LIN {X 0.136,Y -541.302,Z 1152.951,A 0.000,B 0.000,C 90.000,E1 27.078} C_DIS
LIN {X 0.205,Y -536.132,Z 1152.947,A 0.000,B 0.000,C 90.000,E1 26.360} C_DIS
LIN {X 0.131,Y -531.673,Z 1152.943,A 0.000,B 0.000,C 90.000,E1 25.796} C_DIS
LIN {X 0.041,Y -524.620,Z 1152.939,A 0.000,B 0.000,C 90.000,E1 24.951} C_DIS
LIN {X -0.042,Y -515.804,Z 1152.933,A 0.000,B 0.000,C 90.000,E1 23.951} C_DIS
LIN {X -0.075,Y -509.279,Z 1152.929,A 0.000,B 0.000,C 90.000,E1 23.259} C_DIS
LIN {X -0.034,Y -503.804,Z 1152.926,A 0.000,B 0.000,C 90.000,E1 22.695} C_DIS
LIN {X -0.151,Y -492.766,Z 1152.920,A 0.000,B 0.000,C 90.000,E1 21.642} C_DIS
LIN {X -0.103,Y -481.579,Z 1152.914,A 0.000,B 0.000,C 90.000,E1 20.610} C_DIS
LIN {X -0.257,Y -469.838,Z 1152.909,A 0.000,B 0.000,C 90.000,E1 19.577} C_DIS
LIN {X -0.031,Y -457.925,Z 1152.903,A 0.000,B 0.000,C 90.000,E1 18.489} C_DIS
LIN {X -0.234,Y -435.893,Z 1152.891,A 0.000,B 0.000,C 90.000,E1 16.441} C_DIS
LIN {X 0.046,Y -423.104,Z 1152.884,A 0.000,B 0.000,C 90.000,E1 15.064} C_DIS
LIN {X 0.162,Y -412.046,Z 1152.877,A 0.000,B 0.000,C 90.000,E1 13.772} C_DIS
LIN {X 0.036,Y -404.119,Z 1152.871,A 0.000,B 0.000,C 90.000,E1 12.771} C_DIS
LIN {X 0.073,Y -398.095,Z 1152.866,A 0.000,B 0.000,C 90.000,E1 11.895} C_DIS
LIN {X 0.107,Y -396.971,Z 1152.865,A 0.000,B 0.000,C 90.000,E1 11.715} C_DIS
LIN {X -0.009,Y -393.901,Z 1152.862,A 0.000,B 0.000,C 90.000,E1 11.130} C_DIS
LIN {X -0.016,Y -392.561,Z 1152.860,A 0.000,B 0.000,C 90.000,E1 10.715} C_DIS
LIN {X -0.198,Y -392.478,Z 1152.857,A 0.000,B 0.000,C 90.000,E1 10.254} C_DIS
LIN {X 0.110,Y -393.719,Z 1152.853,A 0.000,B 0.000,C 90.000,E1 9.500} C_DIS
LIN {X 0.046,Y -396.236,Z 1152.848,A 0.000,B 0.000,C 90.000,E1 8.624} C_DIS
LIN {X -0.148,Y -401.677,Z 1152.839,A 0.000,B 0.000,C 90.000,E1 7.068} C_DIS
LIN {X -0.013,Y -405.388,Z 1152.835,A 0.000,B 0.000,C 90.000,E1 6.258} C_DIS
LIN {X -0.013,Y -407.563,Z 1152.833,A 0.000,B 0.000,C 90.000,E1 5.910} C_DIS
LIN {X -0.080,Y -410.731,Z 1152.831,A 0.000,B 0.000,C 90.000,E1 5.568} C_DIS
LIN {X 0.043,Y -412.332,Z 1152.830,A 0.000,B 0.000,C 90.000,E1 5.391} C_DIS
LIN {X -0.036,Y -437.093,Z 1152.820,A 0.000,B 0.000,C 90.000,E1 3.555} C_DIS
LIN {X 0.076,Y -456.596,Z 1152.812,A 0.000,B 0.000,C 90.000,E1 2.178} C_DIS
LIN {X -0.104,Y -467.873,Z 1152.808,A 0.000,B 0.000,C 90.000,E1 1.432} C_DIS
LIN {X -0.166,Y -477.392,Z 1152.804,A 0.000,B 0.000,C 90.000,E1 0.802} C_DIS
LIN {X 0.000,Y -488.031,Z 1152.800,A 0.000,B 0.000,C 90.000,E1 360.000} C_DIS
LIN {X 0.105,Y -495.261,Z 1152.797,A 0.000,B 0.000,C 90.000,E1 359.427} C_DIS
LIN {X -0.233,Y -502.565,Z 1152.794,A 0.000,B 0.000,C 90.000,E1 358.854} C_DIS
LIN {X 0.184,Y -509.593,Z 1152.790,A 0.000,B 0.000,C 90.000,E1 358.165} C_DIS
LIN {X 0.238,Y -516.287,Z 1152.786,A 0.000,B 0.000,C 90.000,E1 357.478} C_DIS
LIN {X 0.222,Y -522.608,Z 1152.782,A 0.000,B 0.000,C 90.000,E1 356.788} C_DIS
LIN {X 0.006,Y -528.517,Z 1152.778,A 0.000,B 0.000,C 90.000,E1 356.102} C_DIS
LIN {X -0.016,Y -532.952,Z 1152.775,A 0.000,B 0.000,C 90.000,E1 355.527} C_DIS
LIN {X -0.273,Y -537.881,Z 1152.771,A 0.000,B 0.000,C 90.000,E1 354.837} C_DIS
LIN {X 0.047,Y -542.345,Z 1152.767,A 0.000,B 0.000,C 90.000,E1 354.090} C_DIS
LIN {X 0.129,Y -545.610,Z 1152.764,A 0.000,B 0.000,C 90.000,E1 353.514} C_DIS
LIN {X -0.217,Y -549.964,Z 1152.759,A 0.000,B 0.000,C 90.000,E1 352.704} C_DIS
LIN {X 0.176,Y -552.026,Z 1152.757,A 0.000,B 0.000,C 90.000,E1 352.243} C_DIS
LIN {X 0.150,Y -555.072,Z 1152.753,A 0.000,B 0.000,C 90.000,E1 351.546} C_DIS
LIN {X -0.102,Y -558.385,Z 1152.749,A 0.000,B 0.000,C 90.000,E1 350.735} C_DIS
LIN {X -0.228,Y -561.402,Z 1152.744,A 0.000,B 0.000,C 90.000,E1 349.916} C_DIS
LIN {X -0.261,Y -564.948,Z 1152.738,A 0.000,B 0.000,C 90.000,E1 348.814} C_DIS
LIN {X 0.241,Y -567.386,Z 1152.733,A 0.000,B 0.000,C 90.000,E1 347.937} C_DIS
LIN {X -0.158,Y -570.402,Z 1152.727,A 0.000,B 0.000,C 90.000,E1 346.881} C_DIS
LIN {X -0.189,Y -573.924,Z 1152.719,A 0.000,B 0.000,C 90.000,E1 345.519} C_DIS
LIN {X 0.197,Y -576.570,Z 1152.714,A 0.000,B 0.000,C 90.000,E1 344.393} C_DIS
LIN {X 0.061,Y -579.116,Z 1152.707,A 0.000,B 0.000,C 90.000,E1 343.323} C_DIS
LIN {X 0.129,Y -581.561,Z 1152.701,A 0.000,B 0.000,C 90.000,E1 342.236} C_DIS
LIN {X 0.236,Y -583.874,Z 1152.695,A 0.000,B 0.000,C 90.000,E1 341.148} C_DIS
LIN {X -0.178,Y -585.938,Z 1152.689,A 0.000,B 0.000,C 90.000,E1 340.115} C_DIS
LIN {X 0.319,Y -587.363,Z 1152.685,A 0.000,B 0.000,C 90.000,E1 339.263} C_DIS
LIN {X -0.179,Y -589.454,Z 1152.678,A 0.000,B 0.000,C 90.000,E1 337.975} C_DIS
LIN {X -0.202,Y -590.421,Z 1152.673,A 0.000,B 0.000,C 90.000,E1 337.177} C_DIS
LIN {X 0.343,Y -591.464,Z 1152.666,A 0.000,B 0.000,C 90.000,E1 335.793} C_DIS
LIN {X -0.210,Y -591.834,Z 1152.661,A 0.000,B 0.000,C 90.000,E1 335.049} C_DIS
LIN {X 0.020,Y -591.879,Z 1152.657,A 0.000,B 0.000,C 90.000,E1 334.229} C_DIS
LIN {X 0.081,Y -591.762,Z 1152.654,A 0.000,B 0.000,C 90.000,E1 333.691} C_DIS
LIN {X 0.312,Y -591.168,Z 1152.650,A 0.000,B 0.000,C 90.000,E1 332.871} C_DIS
LIN {X 0.108,Y -590.627,Z 1152.647,A 0.000,B 0.000,C 90.000,E1 332.359} C_DIS
LIN {X 0.073,Y -589.543,Z 1152.642,A 0.000,B 0.000,C 90.000,E1 331.563} C_DIS
LIN {X -0.252,Y -588.050,Z 1152.638,A 0.000,B 0.000,C 90.000,E1 330.795} C_DIS
LIN {X -0.190,Y -586.837,Z 1152.635,A 0.000,B 0.000,C 90.000,E1 330.255} C_DIS
LIN {X 0.248,Y -584.613,Z 1152.630,A 0.000,B 0.000,C 90.000,E1 329.410} C_DIS
LIN {X 0.153,Y -581.952,Z 1152.626,A 0.000,B 0.000,C 90.000,E1 328.614} C_DIS
LIN {X 0.101,Y -579.167,Z 1152.622,A 0.000,B 0.000,C 90.000,E1 327.946} C_DIS
LIN {X 0.330,Y -575.786,Z 1152.618,A 0.000,B 0.000,C 90.000,E1 327.248} C_DIS
LIN {X -0.262,Y -571.745,Z 1152.615,A 0.000,B 0.000,C 90.000,E1 326.628} C_DIS
LIN {X -0.089,Y -567.295,Z 1152.611,A 0.000,B 0.000,C 90.000,E1 325.928} C_DIS
LIN {X -0.172,Y -563.456,Z 1152.608,A 0.000,B 0.000,C 90.000,E1 325.388} C_DIS
LIN {X 0.037,Y -559.163,Z 1152.605,A 0.000,B 0.000,C 90.000,E1 324.815} C_DIS
LIN {X -0.074,Y -551.011,Z 1152.599,A 0.000,B 0.000,C 90.000,E1 323.863} C_DIS
LIN {X 0.078,Y -546.038,Z 1152.596,A 0.000,B 0.000,C 90.000,E1 323.290} C_DIS
LIN {X 0.151,Y -530.643,Z 1152.587,A 0.000,B 0.000,C 90.000,E1 321.618} C_DIS
LIN {X 0.220,Y -526.479,Z 1152.584,A 0.000,B 0.000,C 90.000,E1 321.090} C_DIS
LIN {X 0.001,Y -523.789,Z 1152.581,A 0.000,B 0.000,C 90.000,E1 320.642} C_DIS
LIN {X -0.080,Y -521.477,Z 1152.578,A 0.000,B 0.000,C 90.000,E1 320.070} C_DIS
LIN {X 0.155,Y -520.483,Z 1152.575,A 0.000,B 0.000,C 90.000,E1 319.461} C_DIS
LIN {X -0.167,Y -520.045,Z 1152.570,A 0.000,B 0.000,C 90.000,E1 318.566} C_DIS
LIN {X 0.178,Y -520.307,Z 1152.562,A 0.000,B 0.000,C 90.000,E1 317.067} C_DIS
LIN {X 0.017,Y -521.216,Z 1152.550,A 0.000,B 0.000,C 90.000,E1 315.040} C_DIS
LIN {X 0.024,Y -521.900,Z 1152.542,A 0.000,B 0.000,C 90.000,E1 313.581} C_DIS
LIN {X -0.080,Y -522.795,Z 1152.531,A 0.000,B 0.000,C 90.000,E1 311.553} C_DIS
LIN {X -0.074,Y -523.671,Z 1152.521,A 0.000,B 0.000,C 90.000,E1 309.806} C_DIS
LIN {X 0.307,Y -524.813,Z 1152.510,A 0.000,B 0.000,C 90.000,E1 307.729} C_DIS
LIN {X 0.133,Y -525.768,Z 1152.502,A 0.000,B 0.000,C 90.000,E1 306.297} C_DIS
LIN {X 0.070,Y -526.827,Z 1152.492,A 0.000,B 0.000,C 90.000,E1 304.565} C_DIS
LIN {X 0.067,Y -527.667,Z 1152.484,A 0.000,B 0.000,C 90.000,E1 303.118} C_DIS
LIN {X 0.039,Y -528.892,Z 1152.474,A 0.000,B 0.000,C 90.000,E1 301.386} C_DIS
LIN {X -0.075,Y -530.043,Z 1152.465,A 0.000,B 0.000,C 90.000,E1 299.667} C_DIS
LIN {X -0.250,Y -530.572,Z 1152.460,A 0.000,B 0.000,C 90.000,E1 298.821} C_DIS
LIN {X 0.182,Y -531.222,Z 1152.452,A 0.000,B 0.000,C 90.000,E1 297.334} C_DIS
LIN {X -0.087,Y -531.533,Z 1152.444,A 0.000,B 0.000,C 90.000,E1 295.924} C_DIS
LIN {X 0.126,Y -531.679,Z 1152.436,A 0.000,B 0.000,C 90.000,E1 294.463} C_DIS
LIN {X -0.178,Y -531.663,Z 1152.426,A 0.000,B 0.000,C 90.000,E1 292.770} C_DIS
LIN {X -0.195,Y -531.621,Z 1152.417,A 0.000,B 0.000,C 90.000,E1 291.046} C_DIS
LIN {X 0.089,Y -531.329,Z 1152.409,A 0.000,B 0.000,C 90.000,E1 289.577} C_DIS
LIN {X 0.170,Y -531.006,Z 1152.402,A 0.000,B 0.000,C 90.000,E1 288.417} C_DIS
LIN {X 0.100,Y -530.507,Z 1152.394,A 0.000,B 0.000,C 90.000,E1 286.985} C_DIS
LIN {X 0.198,Y -529.697,Z 1152.385,A 0.000,B 0.000,C 90.000,E1 285.245} C_DIS
LIN {X -0.003,Y -528.817,Z 1152.375,A 0.000,B 0.000,C 90.000,E1 283.536} C_DIS
LIN {X 0.265,Y -527.914,Z 1152.367,A 0.000,B 0.000,C 90.000,E1 282.063} C_DIS
LIN {X -0.094,Y -526.828,Z 1152.358,A 0.000,B 0.000,C 90.000,E1 280.366} C_DIS
LIN {X -0.055,Y -525.829,Z 1152.348,A 0.000,B 0.000,C 90.000,E1 278.624} C_DIS
LIN {X -0.167,Y -524.609,Z 1152.337,A 0.000,B 0.000,C 90.000,E1 276.606} C_DIS
LIN {X -0.255,Y -523.900,Z 1152.329,A 0.000,B 0.000,C 90.000,E1 275.163} C_DIS
LIN {X 0.112,Y -523.232,Z 1152.321,A 0.000,B 0.000,C 90.000,E1 273.669} C_DIS
LIN {X -0.128,Y -522.559,Z 1152.311,A 0.000,B 0.000,C 90.000,E1 271.949} C_DIS
LIN {X 0.187,Y -522.008,Z 1152.303,A 0.000,B 0.000,C 90.000,E1 270.458} C_DIS
LIN {X -0.044,Y -521.317,Z 1152.295,A 0.000,B 0.000,C 90.000,E1 269.026} C_DIS
LIN {X 0.245,Y -520.644,Z 1152.286,A 0.000,B 0.000,C 90.000,E1 267.535} C_DIS
LIN {X 0.056,Y -520.109,Z 1152.280,A 0.000,B 0.000,C 90.000,E1 266.388} C_DIS
LIN {X -0.083,Y -519.632,Z 1152.275,A 0.000,B 0.000,C 90.000,E1 265.527} C_DIS
LIN {X -0.248,Y -518.752,Z 1152.269,A 0.000,B 0.000,C 90.000,E1 264.375} C_DIS
LIN {X 0.089,Y -517.672,Z 1152.262,A 0.000,B 0.000,C 90.000,E1 263.166} C_DIS
LIN {X -0.132,Y -516.199,Z 1152.254,A 0.000,B 0.000,C 90.000,E1 261.724} C_DIS
LIN {X 0.200,Y -514.754,Z 1152.246,A 0.000,B 0.000,C 90.000,E1 260.218} C_DIS
LIN {X 0.008,Y -512.461,Z 1152.233,A 0.000,B 0.000,C 90.000,E1 257.881} C_DIS
LIN {X -0.018,Y -510.366,Z 1152.220,A 0.000,B 0.000,C 90.000,E1 255.519} C_DIS
LIN {X -0.010,Y -508.806,Z 1152.210,A 0.000,B 0.000,C 90.000,E1 253.740} C_DIS
LIN {X 0.189,Y -506.842,Z 1152.198,A 0.000,B 0.000,C 90.000,E1 251.638} C_DIS
LIN {X -0.162,Y -505.371,Z 1152.190,A 0.000,B 0.000,C 90.000,E1 250.188} C_DIS
LIN {X 0.098,Y -503.879,Z 1152.182,A 0.000,B 0.000,C 90.000,E1 248.666} C_DIS
LIN {X 0.120,Y -501.969,Z 1152.172,A 0.000,B 0.000,C 90.000,E1 246.869} C_DIS
LIN {X 0.161,Y -500.575,Z 1152.165,A 0.000,B 0.000,C 90.000,E1 245.665} C_DIS
LIN {X -0.142,Y -498.177,Z 1152.155,A 0.000,B 0.000,C 90.000,E1 243.896} C_DIS
LIN {X 0.114,Y -496.068,Z 1152.147,A 0.000,B 0.000,C 90.000,E1 242.359} C_DIS
LIN {X 0.149,Y -493.416,Z 1152.136,A 0.000,B 0.000,C 90.000,E1 240.539} C_DIS
LIN {X -0.161,Y -492.074,Z 1152.131,A 0.000,B 0.000,C 90.000,E1 239.665} C_DIS
LIN {X 0.276,Y -489.217,Z 1152.121,A 0.000,B 0.000,C 90.000,E1 237.788} C_DIS
LIN {X -0.179,Y -486.354,Z 1152.111,A 0.000,B 0.000,C 90.000,E1 236.008} C_DIS
LIN {X -0.246,Y -483.970,Z 1152.103,A 0.000,B 0.000,C 90.000,E1 234.482} C_DIS
LIN {X 0.101,Y -482.062,Z 1152.096,A 0.000,B 0.000,C 90.000,E1 233.210} C_DIS
LIN {X -0.054,Y -479.043,Z 1152.085,A 0.000,B 0.000,C 90.000,E1 231.376} C_DIS
LIN {X 0.030,Y -477.540,Z 1152.080,A 0.000,B 0.000,C 90.000,E1 230.436} C_DIS
LIN {X 0.287,Y -474.997,Z 1152.072,A 0.000,B 0.000,C 90.000,E1 228.852} C_DIS
LIN {X 0.139,Y -472.390,Z 1152.063,A 0.000,B 0.000,C 90.000,E1 227.310} C_DIS
LIN {X 0.262,Y -469.805,Z 1152.054,A 0.000,B 0.000,C 90.000,E1 225.729} C_DIS
LIN {X -0.095,Y -462.736,Z 1152.023,A 0.000,B 0.000,C 90.000,E1 220.092} C_DIS
LIN {X 0.011,Y -460.932,Z 1152.010,A 0.000,B 0.000,C 90.000,E1 217.855} C_DIS
LIN {X -0.139,Y -459.348,Z 1151.998,A 0.000,B 0.000,C 90.000,E1 215.644} C_DIS
LIN {X -0.208,Y -457.835,Z 1151.970,A 0.000,B 0.000,C 90.000,E1 210.541} C_DIS
LIN {X -0.011,Y -459.088,Z 1151.950,A 0.000,B 0.000,C 90.000,E1 207.001} C_DIS
LIN {X -0.115,Y -461.535,Z 1151.936,A 0.000,B 0.000,C 90.000,E1 204.463} C_DIS
LIN {X -0.027,Y -466.647,Z 1151.918,A 0.000,B 0.000,C 90.000,E1 201.280} C_DIS
LIN {X -0.169,Y -472.328,Z 1151.904,A 0.000,B 0.000,C 90.000,E1 198.779} C_DIS
LIN {X -0.134,Y -480.238,Z 1151.889,A 0.000,B 0.000,C 90.000,E1 195.969} C_DIS
LIN {X 0.189,Y -487.392,Z 1151.877,A 0.000,B 0.000,C 90.000,E1 193.772} C_DIS
LIN {X -0.058,Y -490.516,Z 1151.872,A 0.000,B 0.000,C 90.000,E1 192.883} C_DIS
LIN {X 0.129,Y -499.143,Z 1151.858,A 0.000,B 0.000,C 90.000,E1 190.433} C_DIS
LIN {X 0.196,Y -505.805,Z 1151.848,A 0.000,B 0.000,C 90.000,E1 188.624} C_DIS
LIN {X 0.252,Y -512.574,Z 1151.838,A 0.000,B 0.000,C 90.000,E1 186.834} C_DIS
LIN {X -0.035,Y -518.168,Z 1151.830,A 0.000,B 0.000,C 90.000,E1 185.391} C_DIS
LIN {X 0.246,Y -523.689,Z 1151.822,A 0.000,B 0.000,C 90.000,E1 183.898} C_DIS
LIN {X 0.077,Y -529.165,Z 1151.814,A 0.000,B 0.000,C 90.000,E1 182.465} C_DIS
LIN {X 0.008,Y -534.623,Z 1151.806,A 0.000,B 0.000,C 90.000,E1 181.031} C_DIS
LIN {X 0.027,Y -540.046,Z 1151.798,A 0.000,B 0.000,C 90.000,E1 179.599} C_DIS
LIN {X 0.159,Y -545.569,Z 1151.790,A 0.000,B 0.000,C 90.000,E1 178.165} C_DIS
LIN {X -0.047,Y -553.223,Z 1151.779,A 0.000,B 0.000,C 90.000,E1 176.216} C_DIS
LIN {X -0.199,Y -558.691,Z 1151.771,A 0.000,B 0.000,C 90.000,E1 174.837} C_DIS
LIN {X -0.108,Y -565.163,Z 1151.762,A 0.000,B 0.000,C 90.000,E1 173.166} C_DIS
LIN {X -0.087,Y -569.507,Z 1151.756,A 0.000,B 0.000,C 90.000,E1 172.064} C_DIS
LIN {X 0.108,Y -574.834,Z 1151.748,A 0.000,B 0.000,C 90.000,E1 170.679} C_DIS
LIN {X -0.301,Y -579.038,Z 1151.742,A 0.000,B 0.000,C 90.000,E1 169.634} C_DIS
LIN {X -0.077,Y -585.318,Z 1151.733,A 0.000,B 0.000,C 90.000,E1 167.993} C_DIS
LIN {X -0.232,Y -589.339,Z 1151.727,A 0.000,B 0.000,C 90.000,E1 166.937} C_DIS
LIN {X -0.335,Y -593.227,Z 1151.721,A 0.000,B 0.000,C 90.000,E1 165.880} C_DIS
LIN {X -0.242,Y -596.951,Z 1151.716,A 0.000,B 0.000,C 90.000,E1 164.810} C_DIS
LIN {X -0.094,Y -600.543,Z 1151.710,A 0.000,B 0.000,C 90.000,E1 163.740} C_DIS
LIN {X 0.005,Y -604.837,Z 1151.702,A 0.000,B 0.000,C 90.000,E1 162.417} C_DIS
LIN {X 0.179,Y -608.947,Z 1151.695,A 0.000,B 0.000,C 90.000,E1 161.094} C_DIS
LIN {X -0.214,Y -613.576,Z 1151.686,A 0.000,B 0.000,C 90.000,E1 159.571} C_DIS
LIN {X -0.240,Y -616.490,Z 1151.681,A 0.000,B 0.000,C 90.000,E1 158.539} C_DIS
LIN {X -0.033,Y -620.714,Z 1151.672,A 0.000,B 0.000,C 90.000,E1 156.975} C_DIS
LIN {X 0.268,Y -624.067,Z 1151.665,A 0.000,B 0.000,C 90.000,E1 155.665} C_DIS
LIN {X 0.051,Y -627.391,Z 1151.658,A 0.000,B 0.000,C 90.000,E1 154.409} C_DIS
LIN {X 0.185,Y -631.130,Z 1151.649,A 0.000,B 0.000,C 90.000,E1 152.871} C_DIS
LIN {X -0.209,Y -634.114,Z 1151.642,A 0.000,B 0.000,C 90.000,E1 151.641} C_DIS
LIN {X 0.307,Y -636.973,Z 1151.635,A 0.000,B 0.000,C 90.000,E1 150.333} C_DIS
LIN {X -0.184,Y -640.156,Z 1151.627,A 0.000,B 0.000,C 90.000,E1 148.869} C_DIS
LIN {X 0.211,Y -642.610,Z 1151.620,A 0.000,B 0.000,C 90.000,E1 147.582} C_DIS
LIN {X 0.110,Y -644.885,Z 1151.613,A 0.000,B 0.000,C 90.000,E1 146.342} C_DIS
LIN {X -0.376,Y -646.684,Z 1151.608,A 0.000,B 0.000,C 90.000,E1 145.388} C_DIS
LIN {X 0.007,Y -649.252,Z 1151.599,A 0.000,B 0.000,C 90.000,E1 143.863} C_DIS
LIN {X 0.225,Y -652.104,Z 1151.590,A 0.000,B 0.000,C 90.000,E1 142.110} C_DIS
LIN {X -0.400,Y -655.191,Z 1151.580,A 0.000,B 0.000,C 90.000,E1 140.436} C_DIS
LIN {X -0.084,Y -658.083,Z 1151.572,A 0.000,B 0.000,C 90.000,E1 138.933} C_DIS
LIN {X -0.207,Y -661.090,Z 1151.564,A 0.000,B 0.000,C 90.000,E1 137.472} C_DIS
LIN {X 0.163,Y -664.972,Z 1151.553,A 0.000,B 0.000,C 90.000,E1 135.486} C_DIS
LIN {X 0.168,Y -669.787,Z 1151.541,A 0.000,B 0.000,C 90.000,E1 133.299} C_DIS
LIN {X 0.291,Y -673.754,Z 1151.531,A 0.000,B 0.000,C 90.000,E1 131.595} C_DIS
LIN {X 0.196,Y -678.990,Z 1151.519,A 0.000,B 0.000,C 90.000,E1 129.439} C_DIS
LIN {X 0.012,Y -682.053,Z 1151.513,A 0.000,B 0.000,C 90.000,E1 128.257} C_DIS
LIN {X -0.133,Y -684.994,Z 1151.506,A 0.000,B 0.000,C 90.000,E1 127.076} C_DIS
LIN {X -0.099,Y -688.042,Z 1151.499,A 0.000,B 0.000,C 90.000,E1 125.884} C_DIS
LIN {X 0.022,Y -691.508,Z 1151.491,A 0.000,B 0.000,C 90.000,E1 124.452} C_DIS
LIN {X -0.230,Y -694.370,Z 1151.485,A 0.000,B 0.000,C 90.000,E1 123.293} C_DIS
LIN {X -0.088,Y -696.479,Z 1151.480,A 0.000,B 0.000,C 90.000,E1 122.339} C_DIS
LIN {X 0.058,Y -697.966,Z 1151.476,A 0.000,B 0.000,C 90.000,E1 121.623} C_DIS
LIN {X 0.249,Y -699.712,Z 1151.471,A 0.000,B 0.000,C 90.000,E1 120.669} C_DIS
LIN {X -0.027,Y -703.074,Z 1151.460,A 0.000,B 0.000,C 90.000,E1 118.821} C_DIS
LIN {X 0.198,Y -704.292,Z 1151.456,A 0.000,B 0.000,C 90.000,E1 118.103} C_DIS
LIN {X -0.193,Y -705.284,Z 1151.452,A 0.000,B 0.000,C 90.000,E1 117.436} C_DIS
LIN {X -0.274,Y -705.938,Z 1151.448,A 0.000,B 0.000,C 90.000,E1 116.744} C_DIS
LIN {X 0.247,Y -706.476,Z 1151.442,A 0.000,B 0.000,C 90.000,E1 115.540} C_DIS
LIN {X 0.196,Y -706.527,Z 1151.439,A 0.000,B 0.000,C 90.000,E1 115.079} C_DIS
LIN {X -0.157,Y -706.403,Z 1151.437,A 0.000,B 0.000,C 90.000,E1 114.643} C_DIS
LIN {X 0.135,Y -706.106,Z 1151.436,A 0.000,B 0.000,C 90.000,E1 114.387} C_DIS
LIN {X -0.218,Y -705.160,Z 1151.433,A 0.000,B 0.000,C 90.000,E1 113.951} C_DIS
LIN {X 0.072,Y -703.212,Z 1151.430,A 0.000,B 0.000,C 90.000,E1 113.462} C_DIS
LIN {X -0.291,Y -702.007,Z 1151.429,A 0.000,B 0.000,C 90.000,E1 113.259} C_DIS
LIN {X -0.021,Y -697.617,Z 1151.427,A 0.000,B 0.000,C 90.000,E1 112.770} C_DIS
LIN {X 0.240,Y -696.471,Z 1151.426,A 0.000,B 0.000,C 90.000,E1 112.642} C_DIS
LIN {X -0.143,Y -694.753,Z 1151.425,A 0.000,B 0.000,C 90.000,E1 112.567} C_DIS
LIN {X -0.231,Y -686.248,Z 1151.424,A 0.000,B 0.000,C 90.000,E1 112.280} C_DIS
LIN {X 0.185,Y -684.401,Z 1151.423,A 0.000,B 0.000,C 90.000,E1 112.206} C_DIS
LIN {X 0.091,Y -676.918,Z 1151.423,A 0.000,B 0.000,C 90.000,E1 112.153} C_DIS
LIN {X 0.034,Y -603.707,Z 1151.423,A 0.000,B 0.000,C 90.000,E1 112.153} C_DIS
LIN {X -0.033,Y -600.507,Z 1151.422,A 0.000,B 0.000,C 90.000,E1 111.950} C_DIS
LIN {X 0.099,Y -593.193,Z 1151.419,A 0.000,B 0.000,C 90.000,E1 111.354} C_DIS
LIN {X 0.092,Y -579.957,Z 1151.412,A 0.000,B 0.000,C 90.000,E1 110.194} C_DIS
LIN {X -0.223,Y -574.545,Z 1151.410,A 0.000,B 0.000,C 90.000,E1 109.758} C_DIS
LIN {X 0.062,Y -568.508,Z 1151.407,A 0.000,B 0.000,C 90.000,E1 109.268} C_DIS
LIN {X 0.222,Y -560.556,Z 1151.404,A 0.000,B 0.000,C 90.000,E1 108.725} C_DIS
LIN {X -0.184,Y -555.928,Z 1151.403,A 0.000,B 0.000,C 90.000,E1 108.471} C_DIS
LIN {X 0.243,Y -551.269,Z 1151.401,A 0.000,B 0.000,C 90.000,E1 108.055} C_DIS
LIN {X 0.169,Y -550.152,Z 1151.399,A 0.000,B 0.000,C 90.000,E1 107.873} C_DIS
LIN {X 0.128,Y -550.138,Z 1151.399,A 0.000,B 0.000,C 90.000,E1 107.873} C_DIS
LIN {X 0.049,Y -549.836,Z 1151.397,A 0.000,B 0.000,C 90.000,E1 107.457} C_DIS
LIN {X -0.263,Y -551.058,Z 1151.387,A 0.000,B 0.000,C 90.000,E1 105.607} C_DIS
LIN {X 0.148,Y -552.409,Z 1151.377,A 0.000,B 0.000,C 90.000,E1 103.883} C_DIS
LIN {X -0.210,Y -553.836,Z 1151.368,A 0.000,B 0.000,C 90.000,E1 102.243} C_DIS
LIN {X 0.010,Y -555.406,Z 1151.359,A 0.000,B 0.000,C 90.000,E1 100.546} C_DIS
LIN {X 0.026,Y -556.743,Z 1151.351,A 0.000,B 0.000,C 90.000,E1 99.151} C_DIS
LIN {X 0.257,Y -558.398,Z 1151.340,A 0.000,B 0.000,C 90.000,E1 97.182} C_DIS
LIN {X -0.238,Y -559.663,Z 1151.331,A 0.000,B 0.000,C 90.000,E1 95.568} C_DIS
LIN {X -0.284,Y -560.730,Z 1151.323,A 0.000,B 0.000,C 90.000,E1 94.188} C_DIS
LIN {X -0.222,Y -561.980,Z 1151.314,A 0.000,B 0.000,C 90.000,E1 92.522} C_DIS
LIN {X -0.268,Y -563.062,Z 1151.306,A 0.000,B 0.000,C 90.000,E1 91.146} C_DIS
LIN {X 0.257,Y -564.026,Z 1151.299,A 0.000,B 0.000,C 90.000,E1 89.714} C_DIS
LIN {X 0.232,Y -564.954,Z 1151.291,A 0.000,B 0.000,C 90.000,E1 88.339} C_DIS
LIN {X -0.080,Y -566.057,Z 1151.280,A 0.000,B 0.000,C 90.000,E1 86.445} C_DIS
LIN {X -0.209,Y -567.322,Z 1151.268,A 0.000,B 0.000,C 90.000,E1 84.261} C_DIS
LIN {X 0.208,Y -568.353,Z 1151.257,A 0.000,B 0.000,C 90.000,E1 82.299} C_DIS
LIN {X 0.271,Y -568.933,Z 1151.251,A 0.000,B 0.000,C 90.000,E1 81.197} C_DIS
LIN {X 0.051,Y -569.684,Z 1151.242,A 0.000,B 0.000,C 90.000,E1 79.577} C_DIS
LIN {X 0.231,Y -570.190,Z 1151.236,A 0.000,B 0.000,C 90.000,E1 78.465} C_DIS
LIN {X -0.127,Y -571.119,Z 1151.225,A 0.000,B 0.000,C 90.000,E1 76.589} C_DIS
LIN {X -0.186,Y -572.077,Z 1151.215,A 0.000,B 0.000,C 90.000,E1 74.685} C_DIS
LIN {X -0.221,Y -573.513,Z 1151.201,A 0.000,B 0.000,C 90.000,E1 72.236} C_DIS
LIN {X -0.058,Y -574.874,Z 1151.191,A 0.000,B 0.000,C 90.000,E1 70.315} C_DIS
LIN {X -0.024,Y -576.440,Z 1151.180,A 0.000,B 0.000,C 90.000,E1 68.411} C_DIS
LIN {X 0.272,Y -578.338,Z 1151.170,A 0.000,B 0.000,C 90.000,E1 66.485} C_DIS
LIN {X 0.184,Y -580.302,Z 1151.158,A 0.000,B 0.000,C 90.000,E1 64.332} C_DIS
LIN {X -0.108,Y -581.765,Z 1151.149,A 0.000,B 0.000,C 90.000,E1 62.743} C_DIS
LIN {X -0.117,Y -583.173,Z 1151.140,A 0.000,B 0.000,C 90.000,E1 61.129} C_DIS
LIN {X -0.195,Y -584.249,Z 1151.132,A 0.000,B 0.000,C 90.000,E1 59.793} C_DIS
LIN {X 0.251,Y -585.230,Z 1151.125,A 0.000,B 0.000,C 90.000,E1 58.408} C_DIS
LIN {X -0.289,Y -586.104,Z 1151.117,A 0.000,B 0.000,C 90.000,E1 57.120} C_DIS
LIN {X -0.007,Y -586.926,Z 1151.110,A 0.000,B 0.000,C 90.000,E1 55.754} C_DIS
LIN {X -0.009,Y -587.903,Z 1151.101,A 0.000,B 0.000,C 90.000,E1 54.149} C_DIS
LIN {X -0.115,Y -588.786,Z 1151.092,A 0.000,B 0.000,C 90.000,E1 52.557} C_DIS
LIN {X -0.031,Y -589.506,Z 1151.085,A 0.000,B 0.000,C 90.000,E1 51.215} C_DIS
LIN {X -0.305,Y -590.052,Z 1151.077,A 0.000,B 0.000,C 90.000,E1 49.908} C_DIS
LIN {X 0.044,Y -590.332,Z 1151.071,A 0.000,B 0.000,C 90.000,E1 48.809} C_DIS
LIN {X -0.100,Y -590.481,Z 1151.065,A 0.000,B 0.000,C 90.000,E1 47.757} C_DIS
LIN {X -0.031,Y -590.424,Z 1151.058,A 0.000,B 0.000,C 90.000,E1 46.419} C_DIS
LIN {X 0.272,Y -590.262,Z 1151.052,A 0.000,B 0.000,C 90.000,E1 45.324} C_DIS
LIN {X 0.147,Y -589.950,Z 1151.046,A 0.000,B 0.000,C 90.000,E1 44.271} C_DIS
LIN {X 0.011,Y -589.380,Z 1151.040,A 0.000,B 0.000,C 90.000,E1 43.218} C_DIS
LIN {X -0.350,Y -588.419,Z 1151.033,A 0.000,B 0.000,C 90.000,E1 41.919} C_DIS
LIN {X -0.085,Y -587.318,Z 1151.027,A 0.000,B 0.000,C 90.000,E1 40.825} C_DIS
LIN {X 0.037,Y -586.424,Z 1151.022,A 0.000,B 0.000,C 90.000,E1 40.011} C_DIS
LIN {X 0.069,Y -584.723,Z 1151.015,A 0.000,B 0.000,C 90.000,E1 38.669} C_DIS
LIN {X -0.197,Y -583.551,Z 1151.010,A 0.000,B 0.000,C 90.000,E1 37.890} C_DIS
LIN {X 0.062,Y -581.727,Z 1151.005,A 0.000,B 0.000,C 90.000,E1 36.790} C_DIS
LIN {X -0.229,Y -580.013,Z 1151.000,A 0.000,B 0.000,C 90.000,E1 36.011} C_DIS
LIN {X 0.107,Y -578.819,Z 1150.997,A 0.000,B 0.000,C 90.000,E1 35.438} C_DIS
LIN {X 0.258,Y -576.710,Z 1150.992,A 0.000,B 0.000,C 90.000,E1 34.612} C_DIS
LIN {X -0.087,Y -574.321,Z 1150.988,A 0.000,B 0.000,C 90.000,E1 33.833} C_DIS
LIN {X -0.260,Y -573.501,Z 1150.986,A 0.000,B 0.000,C 90.000,E1 33.579} C_DIS
LIN {X -0.161,Y -570.570,Z 1150.982,A 0.000,B 0.000,C 90.000,E1 32.752} C_DIS
LIN {X -0.096,Y -567.324,Z 1150.977,A 0.000,B 0.000,C 90.000,E1 31.926} C_DIS
LIN {X -0.174,Y -564.942,Z 1150.974,A 0.000,B 0.000,C 90.000,E1 31.386} C_DIS
LIN {X 0.012,Y -561.095,Z 1150.970,A 0.000,B 0.000,C 90.000,E1 30.541} C_DIS
LIN {X -0.045,Y -556.779,Z 1150.965,A 0.000,B 0.000,C 90.000,E1 29.716} C_DIS
LIN {X 0.007,Y -553.712,Z 1150.962,A 0.000,B 0.000,C 90.000,E1 29.155} C_DIS
LIN {X 0.081,Y -548.774,Z 1150.957,A 0.000,B 0.000,C 90.000,E1 28.309} C_DIS
LIN {X -0.027,Y -542.206,Z 1150.952,A 0.000,B 0.000,C 90.000,E1 27.334} C_DIS
LIN {X 0.053,Y -537.217,Z 1150.948,A 0.000,B 0.000,C 90.000,E1 26.616} C_DIS
LIN {X -0.013,Y -532.894,Z 1150.945,A 0.000,B 0.000,C 90.000,E1 26.052} C_DIS
LIN {X -0.177,Y -525.741,Z 1150.940,A 0.000,B 0.000,C 90.000,E1 25.207} C_DIS
LIN {X -0.122,Y -518.293,Z 1150.935,A 0.000,B 0.000,C 90.000,E1 24.335} C_DIS
LIN {X -0.129,Y -514.434,Z 1150.933,A 0.000,B 0.000,C 90.000,E1 23.898} C_DIS
LIN {X -0.277,Y -507.719,Z 1150.929,A 0.000,B 0.000,C 90.000,E1 23.206} C_DIS
LIN {X -0.101,Y -503.603,Z 1150.927,A 0.000,B 0.000,C 90.000,E1 22.770} C_DIS
LIN {X -0.260,Y -493.929,Z 1150.921,A 0.000,B 0.000,C 90.000,E1 21.844} C_DIS
LIN {X 0.212,Y -481.079,Z 1150.915,A 0.000,B 0.000,C 90.000,E1 20.610} C_DIS
LIN {X 0.068,Y -470.770,Z 1150.910,A 0.000,B 0.000,C 90.000,E1 19.704} C_DIS
LIN {X -0.040,Y -458.208,Z 1150.903,A 0.000,B 0.000,C 90.000,E1 18.598} C_DIS
LIN {X -0.108,Y -436.303,Z 1150.892,A 0.000,B 0.000,C 90.000,E1 16.551} C_DIS
LIN {X 0.112,Y -423.551,Z 1150.885,A 0.000,B 0.000,C 90.000,E1 15.190} C_DIS
LIN {X 0.077,Y -412.632,Z 1150.878,A 0.000,B 0.000,C 90.000,E1 13.939} C_DIS
LIN {X 0.136,Y -404.923,Z 1150.872,A 0.000,B 0.000,C 90.000,E1 12.952} C_DIS
LIN {X -0.048,Y -400.070,Z 1150.868,A 0.000,B 0.000,C 90.000,E1 12.299} C_DIS
LIN {X -0.025,Y -396.760,Z 1150.865,A 0.000,B 0.000,C 90.000,E1 11.771} C_DIS
LIN {X 0.132,Y -394.159,Z 1150.863,A 0.000,B 0.000,C 90.000,E1 11.243} C_DIS
LIN {X 0.117,Y -392.536,Z 1150.860,A 0.000,B 0.000,C 90.000,E1 10.725} C_DIS
LIN {X 0.080,Y -392.529,Z 1150.860,A 0.000,B 0.000,C 90.000,E1 10.725} C_DIS
LIN {X -0.025,Y -392.556,Z 1150.857,A 0.000,B 0.000,C 90.000,E1 10.197} C_DIS
LIN {X -0.056,Y -393.416,Z 1150.854,A 0.000,B 0.000,C 90.000,E1 9.670} C_DIS
LIN {X -0.174,Y -396.366,Z 1150.848,A 0.000,B 0.000,C 90.000,E1 8.624} C_DIS
LIN {X 0.081,Y -401.758,Z 1150.839,A 0.000,B 0.000,C 90.000,E1 7.004} C_DIS
LIN {X -0.128,Y -403.966,Z 1150.836,A 0.000,B 0.000,C 90.000,E1 6.543} C_DIS
LIN {X -0.142,Y -405.559,Z 1150.834,A 0.000,B 0.000,C 90.000,E1 6.201} C_DIS
LIN {X 0.076,Y -407.140,Z 1150.833,A 0.000,B 0.000,C 90.000,E1 5.910} C_DIS
LIN {X 0.158,Y -411.590,Z 1150.830,A 0.000,B 0.000,C 90.000,E1 5.391} C_DIS
LIN {X -0.175,Y -417.060,Z 1150.828,A 0.000,B 0.000,C 90.000,E1 4.992} C_DIS
LIN {X 0.001,Y -434.764,Z 1150.820,A 0.000,B 0.000,C 90.000,E1 3.669} C_DIS
LIN {X 0.131,Y -457.555,Z 1150.812,A 0.000,B 0.000,C 90.000,E1 2.064} C_DIS
LIN {X -0.046,Y -467.163,Z 1150.808,A 0.000,B 0.000,C 90.000,E1 1.432} C_DIS
LIN {X -0.161,Y -476.776,Z 1150.804,A 0.000,B 0.000,C 90.000,E1 0.802} C_DIS
LIN {X 0.054,Y -485.912,Z 1150.801,A 0.000,B 0.000,C 90.000,E1 0.115} C_DIS
LIN {X 0.178,Y -491.802,Z 1150.798,A 0.000,B 0.000,C 90.000,E1 359.656} C_DIS
LIN {X 0.076,Y -497.721,Z 1150.796,A 0.000,B 0.000,C 90.000,E1 359.198} C_DIS
LIN {X -0.235,Y -503.562,Z 1150.793,A 0.000,B 0.000,C 90.000,E1 358.740} C_DIS
LIN {X 0.245,Y -510.446,Z 1150.789,A 0.000,B 0.000,C 90.000,E1 358.051} C_DIS
LIN {X -0.224,Y -517.126,Z 1150.786,A 0.000,B 0.000,C 90.000,E1 357.421} C_DIS
LIN {X -0.084,Y -522.319,Z 1150.782,A 0.000,B 0.000,C 90.000,E1 356.846} C_DIS
LIN {X -0.166,Y -528.192,Z 1150.779,A 0.000,B 0.000,C 90.000,E1 356.159} C_DIS
LIN {X -0.190,Y -532.715,Z 1150.775,A 0.000,B 0.000,C 90.000,E1 355.584} C_DIS
LIN {X 0.085,Y -537.712,Z 1150.771,A 0.000,B 0.000,C 90.000,E1 354.837} C_DIS
LIN {X -0.133,Y -542.218,Z 1150.767,A 0.000,B 0.000,C 90.000,E1 354.147} C_DIS
LIN {X -0.053,Y -545.548,Z 1150.764,A 0.000,B 0.000,C 90.000,E1 353.571} C_DIS
LIN {X 0.146,Y -549.944,Z 1150.760,A 0.000,B 0.000,C 90.000,E1 352.704} C_DIS
LIN {X -0.265,Y -552.649,Z 1150.756,A 0.000,B 0.000,C 90.000,E1 352.186} C_DIS
LIN {X -0.033,Y -555.090,Z 1150.753,A 0.000,B 0.000,C 90.000,E1 351.602} C_DIS
LIN {X 0.135,Y -557.421,Z 1150.750,A 0.000,B 0.000,C 90.000,E1 351.027} C_DIS
LIN {X -0.002,Y -560.523,Z 1150.746,A 0.000,B 0.000,C 90.000,E1 350.208} C_DIS
LIN {X -0.203,Y -563.380,Z 1150.741,A 0.000,B 0.000,C 90.000,E1 349.398} C_DIS
LIN {X -0.105,Y -566.766,Z 1150.735,A 0.000,B 0.000,C 90.000,E1 348.285} C_DIS
LIN {X 0.228,Y -570.654,Z 1150.727,A 0.000,B 0.000,C 90.000,E1 346.881} C_DIS
LIN {X 0.203,Y -574.187,Z 1150.720,A 0.000,B 0.000,C 90.000,E1 345.519} C_DIS
LIN {X 0.039,Y -576.859,Z 1150.714,A 0.000,B 0.000,C 90.000,E1 344.448} C_DIS
LIN {X 0.117,Y -580.048,Z 1150.706,A 0.000,B 0.000,C 90.000,E1 343.087} C_DIS
LIN {X -0.145,Y -583.077,Z 1150.699,A 0.000,B 0.000,C 90.000,E1 341.764} C_DIS
LIN {X -0.024,Y -585.316,Z 1150.693,A 0.000,B 0.000,C 90.000,E1 340.678} C_DIS
LIN {X 0.327,Y -587.332,Z 1150.687,A 0.000,B 0.000,C 90.000,E1 339.571} C_DIS
LIN {X -0.171,Y -589.475,Z 1150.679,A 0.000,B 0.000,C 90.000,E1 338.284} C_DIS
LIN {X -0.193,Y -590.604,Z 1150.675,A 0.000,B 0.000,C 90.000,E1 337.486} C_DIS
LIN {X 0.130,Y -591.159,Z 1150.672,A 0.000,B 0.000,C 90.000,E1 336.922} C_DIS
LIN {X 0.014,Y -591.993,Z 1150.666,A 0.000,B 0.000,C 90.000,E1 335.869} C_DIS
LIN {X -0.290,Y -592.412,Z 1150.662,A 0.000,B 0.000,C 90.000,E1 335.101} C_DIS
LIN {X -0.050,Y -592.494,Z 1150.657,A 0.000,B 0.000,C 90.000,E1 334.280} C_DIS
LIN {X -0.244,Y -592.430,Z 1150.654,A 0.000,B 0.000,C 90.000,E1 333.768} C_DIS
LIN {X -0.010,Y -591.884,Z 1150.650,A 0.000,B 0.000,C 90.000,E1 332.948} C_DIS
LIN {X -0.036,Y -591.039,Z 1150.645,A 0.000,B 0.000,C 90.000,E1 332.153} C_DIS
LIN {X -0.346,Y -589.945,Z 1150.641,A 0.000,B 0.000,C 90.000,E1 331.385} C_DIS
LIN {X 0.130,Y -588.375,Z 1150.636,A 0.000,B 0.000,C 90.000,E1 330.539} C_DIS
LIN {X 0.193,Y -587.129,Z 1150.633,A 0.000,B 0.000,C 90.000,E1 329.999} C_DIS
LIN {X 0.250,Y -585.681,Z 1150.630,A 0.000,B 0.000,C 90.000,E1 329.459} C_DIS
LIN {X 0.170,Y -583.092,Z 1150.626,A 0.000,B 0.000,C 90.000,E1 328.663} C_DIS
LIN {X 0.060,Y -579.779,Z 1150.622,A 0.000,B 0.000,C 90.000,E1 327.867} C_DIS
LIN {X -0.015,Y -576.407,Z 1150.618,A 0.000,B 0.000,C 90.000,E1 327.199} C_DIS
LIN {X 0.192,Y -572.415,Z 1150.614,A 0.000,B 0.000,C 90.000,E1 326.501} C_DIS
LIN {X 0.363,Y -567.959,Z 1150.610,A 0.000,B 0.000,C 90.000,E1 325.801} C_DIS
LIN {X -0.184,Y -564.138,Z 1150.607,A 0.000,B 0.000,C 90.000,E1 325.308} C_DIS
LIN {X -0.291,Y -559.875,Z 1150.604,A 0.000,B 0.000,C 90.000,E1 324.769} C_DIS
LIN {X -0.154,Y -551.657,Z 1150.599,A 0.000,B 0.000,C 90.000,E1 323.783} C_DIS
LIN {X -0.031,Y -546.633,Z 1150.596,A 0.000,B 0.000,C 90.000,E1 323.210} C_DIS
LIN {X 0.084,Y -530.152,Z 1150.586,A 0.000,B 0.000,C 90.000,E1 321.412} C_DIS
LIN {X -0.137,Y -526.909,Z 1150.583,A 0.000,B 0.000,C 90.000,E1 321.009} C_DIS
LIN {X 0.004,Y -524.170,Z 1150.581,A 0.000,B 0.000,C 90.000,E1 320.517} C_DIS
LIN {X -0.092,Y -522.113,Z 1150.578,A 0.000,B 0.000,C 90.000,E1 320.033} C_DIS
LIN {X -0.043,Y -520.821,Z 1150.574,A 0.000,B 0.000,C 90.000,E1 319.299} C_DIS
LIN {X 0.274,Y -520.400,Z 1150.568,A 0.000,B 0.000,C 90.000,E1 318.243} C_DIS
LIN {X -0.107,Y -520.678,Z 1150.560,A 0.000,B 0.000,C 90.000,E1 316.824} C_DIS
LIN {X 0.259,Y -521.338,Z 1150.552,A 0.000,B 0.000,C 90.000,E1 315.324} C_DIS
LIN {X 0.260,Y -522.010,Z 1150.544,A 0.000,B 0.000,C 90.000,E1 313.866} C_DIS
LIN {X 0.150,Y -522.864,Z 1150.533,A 0.000,B 0.000,C 90.000,E1 311.838} C_DIS
LIN {X 0.108,Y -523.827,Z 1150.521,A 0.000,B 0.000,C 90.000,E1 309.806} C_DIS
LIN {X -0.169,Y -524.629,Z 1150.513,A 0.000,B 0.000,C 90.000,E1 308.382} C_DIS
LIN {X -0.066,Y -525.718,Z 1150.504,A 0.000,B 0.000,C 90.000,E1 306.629} C_DIS
LIN {X -0.139,Y -526.798,Z 1150.494,A 0.000,B 0.000,C 90.000,E1 304.898} C_DIS
LIN {X 0.143,Y -527.692,Z 1150.486,A 0.000,B 0.000,C 90.000,E1 303.420} C_DIS
LIN {X -0.034,Y -529.046,Z 1150.475,A 0.000,B 0.000,C 90.000,E1 301.416} C_DIS
LIN {X 0.012,Y -529.881,Z 1150.468,A 0.000,B 0.000,C 90.000,E1 300.256} C_DIS
LIN {X -0.041,Y -530.780,Z 1150.460,A 0.000,B 0.000,C 90.000,E1 298.821} C_DIS
LIN {X -0.077,Y -531.469,Z 1150.452,A 0.000,B 0.000,C 90.000,E1 297.385} C_DIS
LIN {X 0.131,Y -531.787,Z 1150.444,A 0.000,B 0.000,C 90.000,E1 295.924} C_DIS
LIN {X 0.157,Y -531.941,Z 1150.438,A 0.000,B 0.000,C 90.000,E1 294.771} C_DIS
LIN {X 0.051,Y -531.965,Z 1150.427,A 0.000,B 0.000,C 90.000,E1 292.770} C_DIS
LIN {X 0.040,Y -531.917,Z 1150.417,A 0.000,B 0.000,C 90.000,E1 291.046} C_DIS
LIN {X -0.171,Y -531.634,Z 1150.409,A 0.000,B 0.000,C 90.000,E1 289.631} C_DIS
LIN {X -0.088,Y -531.334,Z 1150.403,A 0.000,B 0.000,C 90.000,E1 288.471} C_DIS
LIN {X -0.156,Y -530.856,Z 1150.395,A 0.000,B 0.000,C 90.000,E1 287.040} C_DIS
LIN {X -0.054,Y -530.047,Z 1150.385,A 0.000,B 0.000,C 90.000,E1 285.300} C_DIS
LIN {X -0.251,Y -529.156,Z 1150.375,A 0.000,B 0.000,C 90.000,E1 283.592} C_DIS
LIN {X 0.019,Y -528.274,Z 1150.367,A 0.000,B 0.000,C 90.000,E1 282.119} C_DIS
LIN {X 0.209,Y -527.030,Z 1150.356,A 0.000,B 0.000,C 90.000,E1 280.074} C_DIS
LIN {X 0.212,Y -526.402,Z 1150.350,A 0.000,B 0.000,C 90.000,E1 278.916} C_DIS
LIN {X 0.180,Y -525.185,Z 1150.338,A 0.000,B 0.000,C 90.000,E1 276.891} C_DIS
LIN {X 0.048,Y -524.314,Z 1150.329,A 0.000,B 0.000,C 90.000,E1 275.163} C_DIS
LIN {X -0.144,Y -523.537,Z 1150.319,A 0.000,B 0.000,C 90.000,E1 273.440} C_DIS
LIN {X 0.122,Y -522.732,Z 1150.308,A 0.000,B 0.000,C 90.000,E1 271.375} C_DIS
LIN {X -0.053,Y -522.298,Z 1150.301,A 0.000,B 0.000,C 90.000,E1 270.229} C_DIS
LIN {X 0.243,Y -521.574,Z 1150.293,A 0.000,B 0.000,C 90.000,E1 268.740} C_DIS
LIN {X 0.014,Y -520.922,Z 1150.285,A 0.000,B 0.000,C 90.000,E1 267.306} C_DIS
LIN {X -0.193,Y -520.278,Z 1150.277,A 0.000,B 0.000,C 90.000,E1 265.869} C_DIS
LIN {X 0.125,Y -519.424,Z 1150.271,A 0.000,B 0.000,C 90.000,E1 264.666} C_DIS
LIN {X -0.047,Y -518.446,Z 1150.264,A 0.000,B 0.000,C 90.000,E1 263.514} C_DIS
LIN {X -0.273,Y -516.654,Z 1150.254,A 0.000,B 0.000,C 90.000,E1 261.781} C_DIS
LIN {X 0.070,Y -515.206,Z 1150.246,A 0.000,B 0.000,C 90.000,E1 260.274} C_DIS
LIN {X -0.105,Y -512.905,Z 1150.233,A 0.000,B 0.000,C 90.000,E1 257.937} C_DIS
LIN {X -0.149,Y -510.551,Z 1150.218,A 0.000,B 0.000,C 90.000,E1 255.283} C_DIS
LIN {X -0.140,Y -508.919,Z 1150.208,A 0.000,B 0.000,C 90.000,E1 253.504} C_DIS
LIN {X 0.058,Y -507.004,Z 1150.197,A 0.000,B 0.000,C 90.000,E1 251.402} C_DIS
LIN {X -0.030,Y -505.175,Z 1150.187,A 0.000,B 0.000,C 90.000,E1 249.625} C_DIS
LIN {X 0.146,Y -503.988,Z 1150.180,A 0.000,B 0.000,C 90.000,E1 248.411} C_DIS
LIN {X 0.174,Y -501.988,Z 1150.170,A 0.000,B 0.000,C 90.000,E1 246.613} C_DIS
LIN {X 0.218,Y -500.582,Z 1150.164,A 0.000,B 0.000,C 90.000,E1 245.409} C_DIS
LIN {X -0.029,Y -497.754,Z 1150.152,A 0.000,B 0.000,C 90.000,E1 243.332} C_DIS
LIN {X 0.007,Y -495.606,Z 1150.144,A 0.000,B 0.000,C 90.000,E1 241.820} C_DIS
LIN {X 0.301,Y -492.423,Z 1150.132,A 0.000,B 0.000,C 90.000,E1 239.665} C_DIS
LIN {X -0.097,Y -489.106,Z 1150.120,A 0.000,B 0.000,C 90.000,E1 237.582} C_DIS
LIN {X 0.181,Y -485.255,Z 1150.106,A 0.000,B 0.000,C 90.000,E1 235.102} C_DIS
LIN {X -0.094,Y -482.337,Z 1150.096,A 0.000,B 0.000,C 90.000,E1 233.290} C_DIS
LIN {X 0.129,Y -479.288,Z 1150.086,A 0.000,B 0.000,C 90.000,E1 231.412} C_DIS
LIN {X -0.160,Y -477.795,Z 1150.081,A 0.000,B 0.000,C 90.000,E1 230.517} C_DIS
LIN {X 0.102,Y -475.188,Z 1150.072,A 0.000,B 0.000,C 90.000,E1 228.933} C_DIS
LIN {X 0.051,Y -472.069,Z 1150.062,A 0.000,B 0.000,C 90.000,E1 227.067} C_DIS
LIN {X 0.001,Y -468.430,Z 1150.049,A 0.000,B 0.000,C 90.000,E1 224.879} C_DIS
LIN {X -0.261,Y -462.715,Z 1150.023,A 0.000,B 0.000,C 90.000,E1 220.172} C_DIS
LIN {X -0.152,Y -460.807,Z 1150.011,A 0.000,B 0.000,C 90.000,E1 217.935} C_DIS
LIN {X 0.217,Y -459.611,Z 1150.002,A 0.000,B 0.000,C 90.000,E1 216.297} C_DIS
LIN {X -0.146,Y -457.310,Z 1149.970,A 0.000,B 0.000,C 90.000,E1 210.590} C_DIS
LIN {X -0.104,Y -457.875,Z 1149.956,A 0.000,B 0.000,C 90.000,E1 208.025} C_DIS
LIN {X 0.033,Y -459.341,Z 1149.943,A 0.000,B 0.000,C 90.000,E1 205.771} C_DIS
LIN {X -0.103,Y -461.538,Z 1149.933,A 0.000,B 0.000,C 90.000,E1 203.875} C_DIS
LIN {X 0.289,Y -466.401,Z 1149.917,A 0.000,B 0.000,C 90.000,E1 200.972} C_DIS
LIN {X -0.008,Y -472.270,Z 1149.903,A 0.000,B 0.000,C 90.000,E1 198.489} C_DIS
LIN {X 0.173,Y -480.371,Z 1149.887,A 0.000,B 0.000,C 90.000,E1 195.662} C_DIS
LIN {X 0.033,Y -486.590,Z 1149.877,A 0.000,B 0.000,C 90.000,E1 193.828} C_DIS
LIN {X 0.136,Y -490.779,Z 1149.870,A 0.000,B 0.000,C 90.000,E1 192.591} C_DIS
LIN {X -0.070,Y -498.440,Z 1149.858,A 0.000,B 0.000,C 90.000,E1 190.489} C_DIS
LIN {X -0.024,Y -505.120,Z 1149.848,A 0.000,B 0.000,C 90.000,E1 188.681} C_DIS
LIN {X 0.011,Y -511.945,Z 1149.838,A 0.000,B 0.000,C 90.000,E1 186.891} C_DIS
LIN {X 0.224,Y -517.549,Z 1149.830,A 0.000,B 0.000,C 90.000,E1 185.391} C_DIS
LIN {X -0.006,Y -522.017,Z 1149.824,A 0.000,B 0.000,C 90.000,E1 184.245} C_DIS
LIN {X -0.175,Y -527.552,Z 1149.816,A 0.000,B 0.000,C 90.000,E1 182.808} C_DIS
LIN {X 0.245,Y -534.154,Z 1149.806,A 0.000,B 0.000,C 90.000,E1 181.031} C_DIS
LIN {X 0.257,Y -539.639,Z 1149.798,A 0.000,B 0.000,C 90.000,E1 179.599} C_DIS
LIN {X -0.179,Y -545.165,Z 1149.790,A 0.000,B 0.000,C 90.000,E1 178.224} C_DIS
LIN {X 0.172,Y -552.882,Z 1149.779,A 0.000,B 0.000,C 90.000,E1 176.216} C_DIS
LIN {X 0.017,Y -558.439,Z 1149.771,A 0.000,B 0.000,C 90.000,E1 174.837} C_DIS
LIN {X 0.259,Y -566.047,Z 1149.761,A 0.000,B 0.000,C 90.000,E1 172.875} C_DIS
LIN {X 0.220,Y -570.381,Z 1149.755,A 0.000,B 0.000,C 90.000,E1 171.781} C_DIS
LIN {X -0.248,Y -574.721,Z 1149.748,A 0.000,B 0.000,C 90.000,E1 170.735} C_DIS
LIN {X -0.092,Y -578.960,Z 1149.742,A 0.000,B 0.000,C 90.000,E1 169.634} C_DIS
LIN {X 0.134,Y -585.276,Z 1149.733,A 0.000,B 0.000,C 90.000,E1 167.993} C_DIS
LIN {X -0.020,Y -589.333,Z 1149.727,A 0.000,B 0.000,C 90.000,E1 166.937} C_DIS
LIN {X 0.147,Y -594.185,Z 1149.720,A 0.000,B 0.000,C 90.000,E1 165.589} C_DIS
LIN {X -0.027,Y -596.979,Z 1149.716,A 0.000,B 0.000,C 90.000,E1 164.810} C_DIS
LIN {X 0.123,Y -600.572,Z 1149.710,A 0.000,B 0.000,C 90.000,E1 163.740} C_DIS
LIN {X -0.256,Y -604.037,Z 1149.704,A 0.000,B 0.000,C 90.000,E1 162.725} C_DIS
LIN {X 0.168,Y -607.374,Z 1149.698,A 0.000,B 0.000,C 90.000,E1 161.638} C_DIS
LIN {X 0.068,Y -610.563,Z 1149.692,A 0.000,B 0.000,C 90.000,E1 160.604} C_DIS
LIN {X 0.010,Y -613.646,Z 1149.687,A 0.000,B 0.000,C 90.000,E1 159.571} C_DIS
LIN {X -0.044,Y -617.212,Z 1149.679,A 0.000,B 0.000,C 90.000,E1 158.284} C_DIS
LIN {X -0.059,Y -621.447,Z 1149.671,A 0.000,B 0.000,C 90.000,E1 156.741} C_DIS
LIN {X -0.310,Y -626.101,Z 1149.661,A 0.000,B 0.000,C 90.000,E1 154.973} C_DIS
LIN {X 0.319,Y -628.654,Z 1149.655,A 0.000,B 0.000,C 90.000,E1 153.896} C_DIS
LIN {X -0.113,Y -631.741,Z 1149.648,A 0.000,B 0.000,C 90.000,E1 152.666} C_DIS
LIN {X 0.104,Y -635.269,Z 1149.640,A 0.000,B 0.000,C 90.000,E1 151.129} C_DIS
LIN {X 0.081,Y -637.990,Z 1149.633,A 0.000,B 0.000,C 90.000,E1 149.871} C_DIS
LIN {X 0.103,Y -640.584,Z 1149.626,A 0.000,B 0.000,C 90.000,E1 148.614} C_DIS
LIN {X -0.041,Y -643.021,Z 1149.619,A 0.000,B 0.000,C 90.000,E1 147.375} C_DIS
LIN {X -0.081,Y -645.773,Z 1149.610,A 0.000,B 0.000,C 90.000,E1 145.881} C_DIS
LIN {X 0.191,Y -648.781,Z 1149.601,A 0.000,B 0.000,C 90.000,E1 144.116} C_DIS
LIN {X 0.088,Y -651.214,Z 1149.593,A 0.000,B 0.000,C 90.000,E1 142.637} C_DIS
LIN {X -0.166,Y -655.125,Z 1149.580,A 0.000,B 0.000,C 90.000,E1 140.436} C_DIS
LIN {X 0.083,Y -658.993,Z 1149.569,A 0.000,B 0.000,C 90.000,E1 138.447} C_DIS
LIN {X 0.006,Y -661.481,Z 1149.562,A 0.000,B 0.000,C 90.000,E1 137.229} C_DIS
LIN {X 0.395,Y -664.892,Z 1149.553,A 0.000,B 0.000,C 90.000,E1 135.486} C_DIS
LIN {X -0.061,Y -669.685,Z 1149.541,A 0.000,B 0.000,C 90.000,E1 133.338} C_DIS
LIN {X 0.092,Y -674.233,Z 1149.530,A 0.000,B 0.000,C 90.000,E1 131.391} C_DIS
LIN {X 0.451,Y -679.508,Z 1149.518,A 0.000,B 0.000,C 90.000,E1 129.197} C_DIS
LIN {X 0.269,Y -682.580,Z 1149.511,A 0.000,B 0.000,C 90.000,E1 128.016} C_DIS
LIN {X -0.084,Y -686.739,Z 1149.502,A 0.000,B 0.000,C 90.000,E1 126.377} C_DIS
LIN {X -0.015,Y -689.714,Z 1149.495,A 0.000,B 0.000,C 90.000,E1 125.185} C_DIS
LIN {X -0.255,Y -693.178,Z 1149.488,A 0.000,B 0.000,C 90.000,E1 123.785} C_DIS
LIN {X -0.125,Y -695.358,Z 1149.482,A 0.000,B 0.000,C 90.000,E1 122.832} C_DIS
LIN {X 0.035,Y -697.451,Z 1149.477,A 0.000,B 0.000,C 90.000,E1 121.878} C_DIS
LIN {X 0.217,Y -699.231,Z 1149.472,A 0.000,B 0.000,C 90.000,E1 120.924} C_DIS
LIN {X -0.077,Y -702.555,Z 1149.462,A 0.000,B 0.000,C 90.000,E1 119.077} C_DIS
LIN {X -0.198,Y -704.208,Z 1149.456,A 0.000,B 0.000,C 90.000,E1 118.153} C_DIS
LIN {X 0.032,Y -705.213,Z 1149.453,A 0.000,B 0.000,C 90.000,E1 117.436} C_DIS
LIN {X -0.050,Y -705.879,Z 1149.449,A 0.000,B 0.000,C 90.000,E1 116.744} C_DIS
LIN {X 0.176,Y -706.347,Z 1149.443,A 0.000,B 0.000,C 90.000,E1 115.796} C_DIS
LIN {X 0.119,Y -706.505,Z 1149.440,A 0.000,B 0.000,C 90.000,E1 115.103} C_DIS
LIN {X 0.066,Y -706.377,Z 1149.437,A 0.000,B 0.000,C 90.000,E1 114.643} C_DIS
LIN {X 0.357,Y -706.110,Z 1149.436,A 0.000,B 0.000,C 90.000,E1 114.387} C_DIS
LIN {X 0.004,Y -705.207,Z 1149.433,A 0.000,B 0.000,C 90.000,E1 113.951} C_DIS
LIN {X -0.350,Y -703.290,Z 1149.431,A 0.000,B 0.000,C 90.000,E1 113.515} C_DIS
LIN {X -0.070,Y -702.136,Z 1149.429,A 0.000,B 0.000,C 90.000,E1 113.259} C_DIS
LIN {X -0.068,Y -700.021,Z 1149.428,A 0.000,B 0.000,C 90.000,E1 113.025} C_DIS
LIN {X -0.168,Y -696.638,Z 1149.426,A 0.000,B 0.000,C 90.000,E1 112.695} C_DIS
LIN {X -0.163,Y -695.068,Z 1149.425,A 0.000,B 0.000,C 90.000,E1 112.589} C_DIS
LIN {X 0.224,Y -692.649,Z 1149.425,A 0.000,B 0.000,C 90.000,E1 112.461} C_DIS
LIN {X -0.049,Y -686.752,Z 1149.424,A 0.000,B 0.000,C 90.000,E1 112.280} C_DIS
LIN {X 0.282,Y -685.030,Z 1149.424,A 0.000,B 0.000,C 90.000,E1 112.206} C_DIS
LIN {X 0.002,Y -676.431,Z 1149.423,A 0.000,B 0.000,C 90.000,E1 112.153} C_DIS
LIN {X -0.046,Y -603.545,Z 1149.423,A 0.000,B 0.000,C 90.000,E1 112.153} C_DIS
LIN {X 0.306,Y -600.194,Z 1149.422,A 0.000,B 0.000,C 90.000,E1 111.897} C_DIS
LIN {X 0.112,Y -593.199,Z 1149.419,A 0.000,B 0.000,C 90.000,E1 111.354} C_DIS
LIN {X 0.079,Y -579.750,Z 1149.412,A 0.000,B 0.000,C 90.000,E1 110.174} C_DIS
LIN {X -0.012,Y -574.112,Z 1149.410,A 0.000,B 0.000,C 90.000,E1 109.704} C_DIS
LIN {X -0.209,Y -568.101,Z 1149.407,A 0.000,B 0.000,C 90.000,E1 109.268} C_DIS
LIN {X -0.024,Y -560.113,Z 1149.404,A 0.000,B 0.000,C 90.000,E1 108.725} C_DIS
LIN {X 0.042,Y -555.402,Z 1149.402,A 0.000,B 0.000,C 90.000,E1 108.417} C_DIS
LIN {X -0.203,Y -551.410,Z 1149.401,A 0.000,B 0.000,C 90.000,E1 108.127} C_DIS
LIN {X 0.200,Y -550.100,Z 1149.399,A 0.000,B 0.000,C 90.000,E1 107.873} C_DIS
LIN {X 0.157,Y -550.079,Z 1149.399,A 0.000,B 0.000,C 90.000,E1 107.873} C_DIS
LIN {X -0.258,Y -549.819,Z 1149.397,A 0.000,B 0.000,C 90.000,E1 107.457} C_DIS
LIN {X -0.046,Y -551.089,Z 1149.386,A 0.000,B 0.000,C 90.000,E1 105.481} C_DIS
LIN {X -0.192,Y -552.671,Z 1149.375,A 0.000,B 0.000,C 90.000,E1 103.536} C_DIS
LIN {X 0.117,Y -554.126,Z 1149.366,A 0.000,B 0.000,C 90.000,E1 101.827} C_DIS
LIN {X 0.104,Y -555.407,Z 1149.358,A 0.000,B 0.000,C 90.000,E1 100.433} C_DIS
LIN {X 0.213,Y -556.753,Z 1149.350,A 0.000,B 0.000,C 90.000,E1 99.029} C_DIS
LIN {X -0.191,Y -558.399,Z 1149.339,A 0.000,B 0.000,C 90.000,E1 97.125} C_DIS
LIN {X -0.128,Y -559.677,Z 1149.330,A 0.000,B 0.000,C 90.000,E1 95.454} C_DIS
LIN {X -0.259,Y -560.554,Z 1149.324,A 0.000,B 0.000,C 90.000,E1 94.359} C_DIS
LIN {X -0.204,Y -561.833,Z 1149.315,A 0.000,B 0.000,C 90.000,E1 92.694} C_DIS
LIN {X -0.153,Y -563.076,Z 1149.306,A 0.000,B 0.000,C 90.000,E1 91.031} C_DIS
LIN {X -0.191,Y -564.033,Z 1149.298,A 0.000,B 0.000,C 90.000,E1 89.656} C_DIS
LIN {X -0.217,Y -564.951,Z 1149.290,A 0.000,B 0.000,C 90.000,E1 88.282} C_DIS
LIN {X 0.034,Y -566.043,Z 1149.280,A 0.000,B 0.000,C 90.000,E1 86.331} C_DIS
LIN {X -0.204,Y -567.112,Z 1149.269,A 0.000,B 0.000,C 90.000,E1 84.432} C_DIS
LIN {X 0.215,Y -568.135,Z 1149.258,A 0.000,B 0.000,C 90.000,E1 82.470} C_DIS
LIN {X -0.010,Y -568.964,Z 1149.249,A 0.000,B 0.000,C 90.000,E1 80.849} C_DIS
LIN {X 0.059,Y -569.877,Z 1149.239,A 0.000,B 0.000,C 90.000,E1 78.926} C_DIS
LIN {X -0.054,Y -570.586,Z 1149.229,A 0.000,B 0.000,C 90.000,E1 77.297} C_DIS
LIN {X -0.097,Y -571.294,Z 1149.222,A 0.000,B 0.000,C 90.000,E1 75.936} C_DIS
LIN {X 0.041,Y -572.421,Z 1149.210,A 0.000,B 0.000,C 90.000,E1 73.740} C_DIS
LIN {X 0.184,Y -573.634,Z 1149.199,A 0.000,B 0.000,C 90.000,E1 71.819} C_DIS
LIN {X -0.003,Y -575.036,Z 1149.189,A 0.000,B 0.000,C 90.000,E1 69.934} C_DIS
LIN {X -0.324,Y -576.955,Z 1149.177,A 0.000,B 0.000,C 90.000,E1 67.794} C_DIS
LIN {X 0.127,Y -578.528,Z 1149.167,A 0.000,B 0.000,C 90.000,E1 66.125} C_DIS
LIN {X 0.171,Y -580.287,Z 1149.157,A 0.000,B 0.000,C 90.000,E1 64.229} C_DIS
LIN {X 0.129,Y -581.739,Z 1149.148,A 0.000,B 0.000,C 90.000,E1 62.615} C_DIS
LIN {X 0.271,Y -583.340,Z 1149.138,A 0.000,B 0.000,C 90.000,E1 60.717} C_DIS
LIN {X -0.092,Y -584.380,Z 1149.130,A 0.000,B 0.000,C 90.000,E1 59.410} C_DIS
LIN {X -0.150,Y -585.295,Z 1149.123,A 0.000,B 0.000,C 90.000,E1 58.074} C_DIS
LIN {X -0.063,Y -585.991,Z 1149.117,A 0.000,B 0.000,C 90.000,E1 56.993} C_DIS
LIN {X -0.132,Y -586.690,Z 1149.111,A 0.000,B 0.000,C 90.000,E1 55.928} C_DIS
LIN {X 0.074,Y -587.780,Z 1149.100,A 0.000,B 0.000,C 90.000,E1 54.036} C_DIS
LIN {X 0.089,Y -588.626,Z 1149.091,A 0.000,B 0.000,C 90.000,E1 52.431} C_DIS
LIN {X -0.037,Y -589.217,Z 1149.085,A 0.000,B 0.000,C 90.000,E1 51.376} C_DIS
LIN {X 0.313,Y -589.672,Z 1149.079,A 0.000,B 0.000,C 90.000,E1 50.275} C_DIS
LIN {X 0.214,Y -590.018,Z 1149.074,A 0.000,B 0.000,C 90.000,E1 49.218} C_DIS
LIN {X 0.069,Y -590.231,Z 1149.065,A 0.000,B 0.000,C 90.000,E1 47.634} C_DIS
LIN {X 0.124,Y -590.148,Z 1149.057,A 0.000,B 0.000,C 90.000,E1 46.296} C_DIS
LIN {X -0.245,Y -589.900,Z 1149.050,A 0.000,B 0.000,C 90.000,E1 45.000} C_DIS
LIN {X -0.375,Y -589.447,Z 1149.044,A 0.000,B 0.000,C 90.000,E1 43.947} C_DIS
LIN {X 0.156,Y -588.983,Z 1149.040,A 0.000,B 0.000,C 90.000,E1 43.095} C_DIS
LIN {X 0.189,Y -587.976,Z 1149.032,A 0.000,B 0.000,C 90.000,E1 41.757} C_DIS
LIN {X 0.061,Y -586.843,Z 1149.026,A 0.000,B 0.000,C 90.000,E1 40.701} C_DIS
LIN {X -0.080,Y -585.600,Z 1149.020,A 0.000,B 0.000,C 90.000,E1 39.644} C_DIS
LIN {X 0.212,Y -584.180,Z 1149.014,A 0.000,B 0.000,C 90.000,E1 38.543} C_DIS
LIN {X 0.302,Y -583.000,Z 1149.010,A 0.000,B 0.000,C 90.000,E1 37.729} C_DIS
LIN {X 0.199,Y -581.097,Z 1149.004,A 0.000,B 0.000,C 90.000,E1 36.664} C_DIS
LIN {X 0.076,Y -579.982,Z 1149.001,A 0.000,B 0.000,C 90.000,E1 36.137} C_DIS
LIN {X 0.398,Y -577.403,Z 1148.995,A 0.000,B 0.000,C 90.000,E1 35.025} C_DIS
LIN {X 0.060,Y -575.149,Z 1148.990,A 0.000,B 0.000,C 90.000,E1 34.246} C_DIS
LIN {X -0.143,Y -572.569,Z 1148.986,A 0.000,B 0.000,C 90.000,E1 33.452} C_DIS
LIN {X 0.129,Y -570.653,Z 1148.983,A 0.000,B 0.000,C 90.000,E1 32.880} C_DIS
LIN {X 0.072,Y -568.544,Z 1148.980,A 0.000,B 0.000,C 90.000,E1 32.339} C_DIS
LIN {X -0.185,Y -565.064,Z 1148.975,A 0.000,B 0.000,C 90.000,E1 31.544} C_DIS
LIN {X -0.277,Y -562.506,Z 1148.972,A 0.000,B 0.000,C 90.000,E1 31.003} C_DIS
LIN {X 0.094,Y -559.823,Z 1148.969,A 0.000,B 0.000,C 90.000,E1 30.413} C_DIS
LIN {X -0.086,Y -554.730,Z 1148.964,A 0.000,B 0.000,C 90.000,E1 29.461} C_DIS
LIN {X -0.008,Y -549.857,Z 1148.959,A 0.000,B 0.000,C 90.000,E1 28.615} C_DIS
LIN {X 0.126,Y -547.273,Z 1148.957,A 0.000,B 0.000,C 90.000,E1 28.180} C_DIS
LIN {X 0.163,Y -541.653,Z 1148.952,A 0.000,B 0.000,C 90.000,E1 27.334} C_DIS
LIN {X 0.234,Y -536.628,Z 1148.948,A 0.000,B 0.000,C 90.000,E1 26.616} C_DIS
LIN {X 0.023,Y -531.069,Z 1148.944,A 0.000,B 0.000,C 90.000,E1 25.924} C_DIS
LIN {X -0.066,Y -524.011,Z 1148.939,A 0.000,B 0.000,C 90.000,E1 25.079} C_DIS
LIN {X 0.070,Y -516.547,Z 1148.935,A 0.000,B 0.000,C 90.000,E1 24.207} C_DIS
LIN {X 0.163,Y -508.597,Z 1148.930,A 0.000,B 0.000,C 90.000,E1 23.334} C_DIS
LIN {X 0.149,Y -502.984,Z 1148.927,A 0.000,B 0.000,C 90.000,E1 22.770} C_DIS
LIN {X 0.103,Y -496.144,Z 1148.923,A 0.000,B 0.000,C 90.000,E1 22.099} C_DIS
LIN {X 0.009,Y -484.694,Z 1148.917,A 0.000,B 0.000,C 90.000,E1 21.046} C_DIS
LIN {X -0.008,Y -474.367,Z 1148.912,A 0.000,B 0.000,C 90.000,E1 20.120} C_DIS
LIN {X 0.072,Y -464.270,Z 1148.907,A 0.000,B 0.000,C 90.000,E1 19.214} C_DIS
LIN {X -0.134,Y -445.314,Z 1148.897,A 0.000,B 0.000,C 90.000,E1 17.511} C_DIS
LIN {X -0.011,Y -430.899,Z 1148.889,A 0.000,B 0.000,C 90.000,E1 16.079} C_DIS
LIN {X 0.032,Y -416.867,Z 1148.881,A 0.000,B 0.000,C 90.000,E1 14.537} C_DIS
LIN {X -0.127,Y -406.190,Z 1148.874,A 0.000,B 0.000,C 90.000,E1 13.244} C_DIS
LIN {X 0.020,Y -399.885,Z 1148.869,A 0.000,B 0.000,C 90.000,E1 12.355} C_DIS
LIN {X -0.123,Y -396.793,Z 1148.866,A 0.000,B 0.000,C 90.000,E1 11.883} C_DIS
LIN {X 0.046,Y -393.743,Z 1148.863,A 0.000,B 0.000,C 90.000,E1 11.243} C_DIS
LIN {X 0.067,Y -392.437,Z 1148.860,A 0.000,B 0.000,C 90.000,E1 10.725} C_DIS
LIN {X -0.113,Y -392.607,Z 1148.857,A 0.000,B 0.000,C 90.000,E1 10.197} C_DIS
LIN {X -0.144,Y -393.467,Z 1148.854,A 0.000,B 0.000,C 90.000,E1 9.670} C_DIS
LIN {X 0.129,Y -396.435,Z 1148.848,A 0.000,B 0.000,C 90.000,E1 8.568} C_DIS
LIN {X -0.010,Y -401.775,Z 1148.839,A 0.000,B 0.000,C 90.000,E1 7.004} C_DIS
LIN {X 0.135,Y -405.463,Z 1148.834,A 0.000,B 0.000,C 90.000,E1 6.144} C_DIS
LIN {X 0.182,Y -406.796,Z 1148.833,A 0.000,B 0.000,C 90.000,E1 5.910} C_DIS
LIN {X 0.146,Y -409.634,Z 1148.831,A 0.000,B 0.000,C 90.000,E1 5.568} C_DIS
LIN {X -0.122,Y -412.725,Z 1148.829,A 0.000,B 0.000,C 90.000,E1 5.277} C_DIS
LIN {X 0.148,Y -417.991,Z 1148.827,A 0.000,B 0.000,C 90.000,E1 4.821} C_DIS
LIN {X 0.049,Y -427.582,Z 1148.823,A 0.000,B 0.000,C 90.000,E1 4.131} C_DIS
LIN {X -0.011,Y -447.078,Z 1148.815,A 0.000,B 0.000,C 90.000,E1 2.751} C_DIS
LIN {X -0.013,Y -463.149,Z 1148.809,A 0.000,B 0.000,C 90.000,E1 1.661} C_DIS
LIN {X -0.143,Y -476.112,Z 1148.804,A 0.000,B 0.000,C 90.000,E1 0.802} C_DIS
LIN {X 0.217,Y -485.168,Z 1148.801,A 0.000,B 0.000,C 90.000,E1 0.115} C_DIS
LIN {X 0.188,Y -491.343,Z 1148.798,A 0.000,B 0.000,C 90.000,E1 359.656} C_DIS
LIN {X 0.093,Y -497.332,Z 1148.796,A 0.000,B 0.000,C 90.000,E1 359.198} C_DIS
LIN {X -0.086,Y -503.075,Z 1148.793,A 0.000,B 0.000,C 90.000,E1 358.740} C_DIS
LIN {X -0.209,Y -510.158,Z 1148.789,A 0.000,B 0.000,C 90.000,E1 358.108} C_DIS
LIN {X -0.066,Y -516.818,Z 1148.786,A 0.000,B 0.000,C 90.000,E1 357.421} C_DIS
LIN {X -0.249,Y -521.859,Z 1148.783,A 0.000,B 0.000,C 90.000,E1 356.906} C_DIS
LIN {X 0.006,Y -528.011,Z 1148.779,A 0.000,B 0.000,C 90.000,E1 356.159} C_DIS
LIN {X -0.019,Y -532.613,Z 1148.776,A 0.000,B 0.000,C 90.000,E1 355.584} C_DIS
LIN {X 0.257,Y -537.661,Z 1148.771,A 0.000,B 0.000,C 90.000,E1 354.837} C_DIS
LIN {X 0.041,Y -542.209,Z 1148.768,A 0.000,B 0.000,C 90.000,E1 354.147} C_DIS
LIN {X 0.121,Y -545.584,Z 1148.764,A 0.000,B 0.000,C 90.000,E1 353.571} C_DIS
LIN {X -0.224,Y -550.016,Z 1148.760,A 0.000,B 0.000,C 90.000,E1 352.761} C_DIS
LIN {X -0.088,Y -552.743,Z 1148.757,A 0.000,B 0.000,C 90.000,E1 352.186} C_DIS
LIN {X 0.188,Y -556.395,Z 1148.752,A 0.000,B 0.000,C 90.000,E1 351.319} C_DIS
LIN {X -0.102,Y -558.637,Z 1148.749,A 0.000,B 0.000,C 90.000,E1 350.792} C_DIS
LIN {X 0.231,Y -561.694,Z 1148.744,A 0.000,B 0.000,C 90.000,E1 349.926} C_DIS
LIN {X 0.142,Y -564.474,Z 1148.740,A 0.000,B 0.000,C 90.000,E1 349.106} C_DIS
LIN {X 0.086,Y -566.993,Z 1148.735,A 0.000,B 0.000,C 90.000,E1 348.285} C_DIS
LIN {X 0.240,Y -570.158,Z 1148.729,A 0.000,B 0.000,C 90.000,E1 347.173} C_DIS
LIN {X 0.242,Y -572.388,Z 1148.724,A 0.000,B 0.000,C 90.000,E1 346.353} C_DIS
LIN {X 0.247,Y -575.869,Z 1148.717,A 0.000,B 0.000,C 90.000,E1 344.991} C_DIS
LIN {X -0.104,Y -577.818,Z 1148.712,A 0.000,B 0.000,C 90.000,E1 344.212} C_DIS
LIN {X -0.014,Y -581.034,Z 1148.705,A 0.000,B 0.000,C 90.000,E1 342.851} C_DIS
LIN {X 0.078,Y -583.471,Z 1148.699,A 0.000,B 0.000,C 90.000,E1 341.764} C_DIS
LIN {X 0.204,Y -585.745,Z 1148.693,A 0.000,B 0.000,C 90.000,E1 340.678} C_DIS
LIN {X 0.227,Y -588.230,Z 1148.685,A 0.000,B 0.000,C 90.000,E1 339.337} C_DIS
LIN {X -0.043,Y -590.367,Z 1148.678,A 0.000,B 0.000,C 90.000,E1 338.028} C_DIS
LIN {X -0.054,Y -591.407,Z 1148.673,A 0.000,B 0.000,C 90.000,E1 337.230} C_DIS
LIN {X -0.061,Y -592.100,Z 1148.669,A 0.000,B 0.000,C 90.000,E1 336.433} C_DIS
LIN {X 0.173,Y -592.720,Z 1148.665,A 0.000,B 0.000,C 90.000,E1 335.613} C_DIS
LIN {X -0.120,Y -593.096,Z 1148.660,A 0.000,B 0.000,C 90.000,E1 334.845} C_DIS
LIN {X 0.128,Y -593.120,Z 1148.656,A 0.000,B 0.000,C 90.000,E1 334.024} C_DIS
LIN {X -0.063,Y -592.966,Z 1148.653,A 0.000,B 0.000,C 90.000,E1 333.512} C_DIS
LIN {X 0.177,Y -592.375,Z 1148.648,A 0.000,B 0.000,C 90.000,E1 332.692} C_DIS
LIN {X 0.155,Y -591.488,Z 1148.644,A 0.000,B 0.000,C 90.000,E1 331.897} C_DIS
LIN {X -0.151,Y -590.336,Z 1148.640,A 0.000,B 0.000,C 90.000,E1 331.129} C_DIS
LIN {X -0.186,Y -588.689,Z 1148.635,A 0.000,B 0.000,C 90.000,E1 330.333} C_DIS
LIN {X -0.236,Y -586.643,Z 1148.631,A 0.000,B 0.000,C 90.000,E1 329.537} C_DIS
LIN {X -0.180,Y -585.011,Z 1148.628,A 0.000,B 0.000,C 90.000,E1 328.997} C_DIS
LIN {X -0.133,Y -583.104,Z 1148.625,A 0.000,B 0.000,C 90.000,E1 328.456} C_DIS
LIN {X -0.169,Y -580.297,Z 1148.621,A 0.000,B 0.000,C 90.000,E1 327.788} C_DIS
LIN {X -0.236,Y -576.944,Z 1148.617,A 0.000,B 0.000,C 90.000,E1 327.120} C_DIS
LIN {X -0.022,Y -572.978,Z 1148.614,A 0.000,B 0.000,C 90.000,E1 326.421} C_DIS
LIN {X 0.159,Y -568.538,Z 1148.610,A 0.000,B 0.000,C 90.000,E1 325.722} C_DIS
LIN {X 0.083,Y -564.679,Z 1148.607,A 0.000,B 0.000,C 90.000,E1 325.182} C_DIS
LIN {X 0.084,Y -561.585,Z 1148.604,A 0.000,B 0.000,C 90.000,E1 324.769} C_DIS
LIN {X 0.362,Y -554.661,Z 1148.600,A 0.000,B 0.000,C 90.000,E1 323.909} C_DIS
LIN {X -0.200,Y -547.176,Z 1148.595,A 0.000,B 0.000,C 90.000,E1 323.130} C_DIS
LIN {X -0.140,Y -534.344,Z 1148.587,A 0.000,B 0.000,C 90.000,E1 321.743} C_DIS
LIN {X -0.188,Y -530.689,Z 1148.585,A 0.000,B 0.000,C 90.000,E1 321.331} C_DIS
LIN {X -0.174,Y -527.840,Z 1148.583,A 0.000,B 0.000,C 90.000,E1 320.964} C_DIS
LIN {X -0.109,Y -524.980,Z 1148.580,A 0.000,B 0.000,C 90.000,E1 320.481} C_DIS
LIN {X 0.020,Y -522.897,Z 1148.578,A 0.000,B 0.000,C 90.000,E1 319.989} C_DIS
LIN {X 0.141,Y -521.618,Z 1148.574,A 0.000,B 0.000,C 90.000,E1 319.380} C_DIS
LIN {X -0.054,Y -521.336,Z 1148.574,A 0.000,B 0.000,C 90.000,E1 319.256} C_DIS
LIN {X -0.126,Y -520.771,Z 1148.568,A 0.000,B 0.000,C 90.000,E1 318.243} C_DIS
LIN {X -0.345,Y -520.804,Z 1148.563,A 0.000,B 0.000,C 90.000,E1 317.391} C_DIS
LIN {X -0.130,Y -521.630,Z 1148.552,A 0.000,B 0.000,C 90.000,E1 315.324} C_DIS
LIN {X -0.122,Y -522.266,Z 1148.544,A 0.000,B 0.000,C 90.000,E1 313.866} C_DIS
LIN {X -0.228,Y -523.064,Z 1148.532,A 0.000,B 0.000,C 90.000,E1 311.838} C_DIS
LIN {X -0.178,Y -523.718,Z 1148.524,A 0.000,B 0.000,C 90.000,E1 310.378} C_DIS
LIN {X -0.090,Y -524.667,Z 1148.515,A 0.000,B 0.000,C 90.000,E1 308.624} C_DIS
LIN {X 0.022,Y -525.720,Z 1148.505,A 0.000,B 0.000,C 90.000,E1 306.870} C_DIS
LIN {X 0.261,Y -526.818,Z 1148.495,A 0.000,B 0.000,C 90.000,E1 305.105} C_DIS
LIN {X -0.186,Y -527.760,Z 1148.487,A 0.000,B 0.000,C 90.000,E1 303.706} C_DIS
LIN {X -0.114,Y -529.249,Z 1148.474,A 0.000,B 0.000,C 90.000,E1 301.386} C_DIS
LIN {X 0.117,Y -530.103,Z 1148.468,A 0.000,B 0.000,C 90.000,E1 300.207} C_DIS
LIN {X 0.076,Y -531.026,Z 1148.460,A 0.000,B 0.000,C 90.000,E1 298.771} C_DIS
LIN {X 0.051,Y -531.737,Z 1148.452,A 0.000,B 0.000,C 90.000,E1 297.334} C_DIS
LIN {X 0.024,Y -532.056,Z 1148.444,A 0.000,B 0.000,C 90.000,E1 295.899} C_DIS
LIN {X -0.180,Y -532.201,Z 1148.438,A 0.000,B 0.000,C 90.000,E1 294.771} C_DIS
LIN {X 0.016,Y -532.251,Z 1148.428,A 0.000,B 0.000,C 90.000,E1 293.025} C_DIS
LIN {X 0.209,Y -532.223,Z 1148.418,A 0.000,B 0.000,C 90.000,E1 291.280} C_DIS
LIN {X 0.110,Y -532.096,Z 1148.414,A 0.000,B 0.000,C 90.000,E1 290.429} C_DIS
LIN {X -0.105,Y -531.797,Z 1148.406,A 0.000,B 0.000,C 90.000,E1 289.014} C_DIS
LIN {X 0.017,Y -531.298,Z 1148.396,A 0.000,B 0.000,C 90.000,E1 287.275} C_DIS
LIN {X -0.015,Y -530.485,Z 1148.386,A 0.000,B 0.000,C 90.000,E1 285.552} C_DIS
LIN {X -0.062,Y -529.641,Z 1148.377,A 0.000,B 0.000,C 90.000,E1 283.828} C_DIS
LIN {X 0.250,Y -528.578,Z 1148.367,A 0.000,B 0.000,C 90.000,E1 282.063} C_DIS
LIN {X -0.095,Y -527.546,Z 1148.358,A 0.000,B 0.000,C 90.000,E1 280.366} C_DIS
LIN {X -0.060,Y -526.746,Z 1148.349,A 0.000,B 0.000,C 90.000,E1 278.916} C_DIS
LIN {X -0.083,Y -525.563,Z 1148.338,A 0.000,B 0.000,C 90.000,E1 276.891} C_DIS
LIN {X -0.206,Y -524.681,Z 1148.329,A 0.000,B 0.000,C 90.000,E1 275.163} C_DIS
LIN {X 0.120,Y -523.815,Z 1148.317,A 0.000,B 0.000,C 90.000,E1 273.094} C_DIS
LIN {X -0.114,Y -523.112,Z 1148.308,A 0.000,B 0.000,C 90.000,E1 271.375} C_DIS
LIN {X 0.197,Y -522.545,Z 1148.300,A 0.000,B 0.000,C 90.000,E1 269.885} C_DIS
LIN {X -0.153,Y -521.426,Z 1148.287,A 0.000,B 0.000,C 90.000,E1 267.593} C_DIS
LIN {X 0.116,Y -520.647,Z 1148.277,A 0.000,B 0.000,C 90.000,E1 265.812} C_DIS
LIN {X -0.079,Y -519.813,Z 1148.270,A 0.000,B 0.000,C 90.000,E1 264.666} C_DIS
LIN {X -0.174,Y -519.134,Z 1148.266,A 0.000,B 0.000,C 90.000,E1 263.799} C_DIS
LIN {X 0.138,Y -517.348,Z 1148.256,A 0.000,B 0.000,C 90.000,E1 262.008} C_DIS
LIN {X -0.110,Y -515.583,Z 1148.246,A 0.000,B 0.000,C 90.000,E1 260.274} C_DIS
LIN {X -0.250,Y -513.532,Z 1148.234,A 0.000,B 0.000,C 90.000,E1 258.229} C_DIS
LIN {X 0.232,Y -512.143,Z 1148.226,A 0.000,B 0.000,C 90.000,E1 256.700} C_DIS
LIN {X 0.189,Y -510.894,Z 1148.218,A 0.000,B 0.000,C 90.000,E1 255.227} C_DIS
LIN {X -0.288,Y -509.272,Z 1148.208,A 0.000,B 0.000,C 90.000,E1 253.504} C_DIS
LIN {X -0.081,Y -507.345,Z 1148.197,A 0.000,B 0.000,C 90.000,E1 251.402} C_DIS
LIN {X 0.222,Y -505.812,Z 1148.188,A 0.000,B 0.000,C 90.000,E1 249.880} C_DIS
LIN {X 0.021,Y -504.303,Z 1148.180,A 0.000,B 0.000,C 90.000,E1 248.411} C_DIS
LIN {X 0.057,Y -502.288,Z 1148.170,A 0.000,B 0.000,C 90.000,E1 246.613} C_DIS
LIN {X 0.105,Y -500.872,Z 1148.163,A 0.000,B 0.000,C 90.000,E1 245.409} C_DIS
LIN {X -0.134,Y -498.037,Z 1148.152,A 0.000,B 0.000,C 90.000,E1 243.332} C_DIS
LIN {X -0.091,Y -495.877,Z 1148.143,A 0.000,B 0.000,C 90.000,E1 241.820} C_DIS
LIN {X 0.210,Y -492.658,Z 1148.132,A 0.000,B 0.000,C 90.000,E1 239.665} C_DIS
LIN {X -0.182,Y -489.331,Z 1148.120,A 0.000,B 0.000,C 90.000,E1 237.582} C_DIS
LIN {X 0.276,Y -485.936,Z 1148.108,A 0.000,B 0.000,C 90.000,E1 235.388} C_DIS
LIN {X 0.013,Y -483.030,Z 1148.098,A 0.000,B 0.000,C 90.000,E1 233.577} C_DIS
LIN {X 0.063,Y -480.436,Z 1148.089,A 0.000,B 0.000,C 90.000,E1 232.029} C_DIS
LIN {X -0.226,Y -477.925,Z 1148.081,A 0.000,B 0.000,C 90.000,E1 230.517} C_DIS
LIN {X 0.037,Y -475.271,Z 1148.072,A 0.000,B 0.000,C 90.000,E1 228.933} C_DIS
LIN {X -0.012,Y -472.154,Z 1148.062,A 0.000,B 0.000,C 90.000,E1 227.067} C_DIS
LIN {X 0.052,Y -465.778,Z 1148.039,A 0.000,B 0.000,C 90.000,E1 222.975} C_DIS
LIN {X -0.118,Y -463.272,Z 1148.026,A 0.000,B 0.000,C 90.000,E1 220.782} C_DIS
LIN {X 0.265,Y -461.466,Z 1148.016,A 0.000,B 0.000,C 90.000,E1 218.830} C_DIS
LIN {X -0.231,Y -459.645,Z 1148.004,A 0.000,B 0.000,C 90.000,E1 216.664} C_DIS
LIN {X 0.158,Y -456.792,Z 1147.970,A 0.000,B 0.000,C 90.000,E1 210.541} C_DIS
LIN {X 0.085,Y -457.053,Z 1147.957,A 0.000,B 0.000,C 90.000,E1 208.309} C_DIS
LIN {X -0.092,Y -458.569,Z 1147.943,A 0.000,B 0.000,C 90.000,E1 205.771} C_DIS
LIN {X 0.091,Y -461.199,Z 1147.931,A 0.000,B 0.000,C 90.000,E1 203.515} C_DIS
LIN {X 0.115,Y -465.621,Z 1147.917,A 0.000,B 0.000,C 90.000,E1 200.972} C_DIS
LIN {X -0.009,Y -470.707,Z 1147.904,A 0.000,B 0.000,C 90.000,E1 198.779} C_DIS
LIN {X 0.170,Y -476.802,Z 1147.892,A 0.000,B 0.000,C 90.000,E1 196.567} C_DIS
LIN {X -0.214,Y -485.990,Z 1147.877,A 0.000,B 0.000,C 90.000,E1 193.828} C_DIS
LIN {X -0.122,Y -490.239,Z 1147.870,A 0.000,B 0.000,C 90.000,E1 192.591} C_DIS
LIN {X 0.145,Y -497.949,Z 1147.858,A 0.000,B 0.000,C 90.000,E1 190.433} C_DIS
LIN {X 0.184,Y -504.669,Z 1147.848,A 0.000,B 0.000,C 90.000,E1 188.624} C_DIS
LIN {X -0.244,Y -510.406,Z 1147.840,A 0.000,B 0.000,C 90.000,E1 187.182} C_DIS
LIN {X -0.056,Y -516.058,Z 1147.832,A 0.000,B 0.000,C 90.000,E1 185.682} C_DIS
LIN {X 0.192,Y -521.673,Z 1147.823,A 0.000,B 0.000,C 90.000,E1 184.188} C_DIS
LIN {X 0.020,Y -527.258,Z 1147.815,A 0.000,B 0.000,C 90.000,E1 182.751} C_DIS
LIN {X -0.098,Y -533.921,Z 1147.806,A 0.000,B 0.000,C 90.000,E1 181.031} C_DIS
LIN {X -0.094,Y -539.468,Z 1147.798,A 0.000,B 0.000,C 90.000,E1 179.599} C_DIS
LIN {X 0.060,Y -546.112,Z 1147.788,A 0.000,B 0.000,C 90.000,E1 177.879} C_DIS
LIN {X -0.193,Y -552.782,Z 1147.779,A 0.000,B 0.000,C 90.000,E1 176.216} C_DIS
LIN {X -0.231,Y -559.497,Z 1147.770,A 0.000,B 0.000,C 90.000,E1 174.546} C_DIS
LIN {X -0.116,Y -566.103,Z 1147.760,A 0.000,B 0.000,C 90.000,E1 172.875} C_DIS
LIN {X 0.209,Y -572.672,Z 1147.751,A 0.000,B 0.000,C 90.000,E1 171.197} C_DIS
LIN {X -0.014,Y -578.071,Z 1147.744,A 0.000,B 0.000,C 90.000,E1 169.859} C_DIS
LIN {X -0.249,Y -585.459,Z 1147.733,A 0.000,B 0.000,C 90.000,E1 167.993} C_DIS
LIN {X -0.145,Y -590.514,Z 1147.726,A 0.000,B 0.000,C 90.000,E1 166.645} C_DIS
LIN {X -0.087,Y -594.423,Z 1147.720,A 0.000,B 0.000,C 90.000,E1 165.574} C_DIS
LIN {X 0.319,Y -599.034,Z 1147.713,A 0.000,B 0.000,C 90.000,E1 164.212} C_DIS
LIN {X 0.220,Y -603.418,Z 1147.705,A 0.000,B 0.000,C 90.000,E1 162.906} C_DIS
LIN {X 0.060,Y -606.786,Z 1147.699,A 0.000,B 0.000,C 90.000,E1 161.873} C_DIS
LIN {X 0.265,Y -610.772,Z 1147.692,A 0.000,B 0.000,C 90.000,E1 160.550} C_DIS
LIN {X 0.208,Y -613.850,Z 1147.686,A 0.000,B 0.000,C 90.000,E1 159.518} C_DIS
LIN {X 0.153,Y -617.391,Z 1147.679,A 0.000,B 0.000,C 90.000,E1 158.230} C_DIS
LIN {X -0.180,Y -620.926,Z 1147.672,A 0.000,B 0.000,C 90.000,E1 156.975} C_DIS
LIN {X -0.125,Y -625.605,Z 1147.662,A 0.000,B 0.000,C 90.000,E1 155.177} C_DIS
LIN {X -0.073,Y -628.175,Z 1147.656,A 0.000,B 0.000,C 90.000,E1 154.152} C_DIS
LIN {X 0.075,Y -631.862,Z 1147.648,A 0.000,B 0.000,C 90.000,E1 152.615} C_DIS
LIN {X -0.269,Y -635.357,Z 1147.640,A 0.000,B 0.000,C 90.000,E1 151.129} C_DIS
LIN {X -0.291,Y -638.055,Z 1147.633,A 0.000,B 0.000,C 90.000,E1 149.871} C_DIS
LIN {X 0.116,Y -641.135,Z 1147.624,A 0.000,B 0.000,C 90.000,E1 148.329} C_DIS
LIN {X -0.361,Y -643.555,Z 1147.617,A 0.000,B 0.000,C 90.000,E1 147.120} C_DIS
LIN {X -0.093,Y -645.808,Z 1147.610,A 0.000,B 0.000,C 90.000,E1 145.849} C_DIS
LIN {X -0.185,Y -648.806,Z 1147.601,A 0.000,B 0.000,C 90.000,E1 144.116} C_DIS
LIN {X -0.289,Y -651.243,Z 1147.592,A 0.000,B 0.000,C 90.000,E1 142.637} C_DIS
LIN {X 0.379,Y -655.156,Z 1147.580,A 0.000,B 0.000,C 90.000,E1 140.356} C_DIS
LIN {X 0.197,Y -659.004,Z 1147.569,A 0.000,B 0.000,C 90.000,E1 138.405} C_DIS
LIN {X -0.375,Y -661.487,Z 1147.562,A 0.000,B 0.000,C 90.000,E1 137.229} C_DIS
LIN {X 0.012,Y -664.910,Z 1147.553,A 0.000,B 0.000,C 90.000,E1 135.486} C_DIS
LIN {X 0.014,Y -669.702,Z 1147.541,A 0.000,B 0.000,C 90.000,E1 133.299} C_DIS
LIN {X 0.150,Y -674.256,Z 1147.530,A 0.000,B 0.000,C 90.000,E1 131.353} C_DIS
LIN {X -0.100,Y -677.685,Z 1147.522,A 0.000,B 0.000,C 90.000,E1 129.930} C_DIS
LIN {X 0.246,Y -681.383,Z 1147.514,A 0.000,B 0.000,C 90.000,E1 128.463} C_DIS
LIN {X 0.059,Y -683.770,Z 1147.509,A 0.000,B 0.000,C 90.000,E1 127.523} C_DIS
LIN {X -0.069,Y -686.769,Z 1147.502,A 0.000,B 0.000,C 90.000,E1 126.343} C_DIS
LIN {X -0.010,Y -689.752,Z 1147.495,A 0.000,B 0.000,C 90.000,E1 125.152} C_DIS
LIN {X 0.313,Y -693.229,Z 1147.487,A 0.000,B 0.000,C 90.000,E1 123.706} C_DIS
LIN {X -0.143,Y -695.385,Z 1147.482,A 0.000,B 0.000,C 90.000,E1 122.801} C_DIS
LIN {X -0.360,Y -697.489,Z 1147.477,A 0.000,B 0.000,C 90.000,E1 121.878} C_DIS
LIN {X -0.180,Y -699.264,Z 1147.472,A 0.000,B 0.000,C 90.000,E1 120.924} C_DIS
LIN {X -0.198,Y -703.002,Z 1147.460,A 0.000,B 0.000,C 90.000,E1 118.821} C_DIS
LIN {X 0.025,Y -704.214,Z 1147.456,A 0.000,B 0.000,C 90.000,E1 118.103} C_DIS
LIN {X 0.260,Y -705.192,Z 1147.452,A 0.000,B 0.000,C 90.000,E1 117.385} C_DIS
LIN {X 0.182,Y -705.843,Z 1147.448,A 0.000,B 0.000,C 90.000,E1 116.693} C_DIS
LIN {X -0.222,Y -706.322,Z 1147.443,A 0.000,B 0.000,C 90.000,E1 115.796} C_DIS
LIN {X 0.019,Y -706.466,Z 1147.439,A 0.000,B 0.000,C 90.000,E1 115.079} C_DIS
LIN {X -0.334,Y -706.341,Z 1147.437,A 0.000,B 0.000,C 90.000,E1 114.643} C_DIS
LIN {X -0.041,Y -705.580,Z 1147.434,A 0.000,B 0.000,C 90.000,E1 114.155} C_DIS
LIN {X 0.250,Y -705.113,Z 1147.433,A 0.000,B 0.000,C 90.000,E1 113.898} C_DIS
LIN {X 0.037,Y -702.637,Z 1147.430,A 0.000,B 0.000,C 90.000,E1 113.334} C_DIS
LIN {X 0.176,Y -701.898,Z 1147.429,A 0.000,B 0.000,C 90.000,E1 113.206} C_DIS
LIN {X -0.181,Y -697.374,Z 1147.427,A 0.000,B 0.000,C 90.000,E1 112.770} C_DIS
LIN {X -0.046,Y -696.017,Z 1147.426,A 0.000,B 0.000,C 90.000,E1 112.642} C_DIS
LIN {X 0.085,Y -693.802,Z 1147.425,A 0.000,B 0.000,C 90.000,E1 112.514} C_DIS
LIN {X 0.399,Y -685.550,Z 1147.424,A 0.000,B 0.000,C 90.000,E1 112.206} C_DIS
LIN {X 0.148,Y -684.424,Z 1147.423,A 0.000,B 0.000,C 90.000,E1 112.206} C_DIS
LIN {X -0.008,Y -676.936,Z 1147.423,A 0.000,B 0.000,C 90.000,E1 112.153} C_DIS
LIN {X -0.054,Y -603.495,Z 1147.423,A 0.000,B 0.000,C 90.000,E1 112.153} C_DIS
LIN {X -0.175,Y -600.245,Z 1147.422,A 0.000,B 0.000,C 90.000,E1 111.950} C_DIS
LIN {X -0.176,Y -595.604,Z 1147.420,A 0.000,B 0.000,C 90.000,E1 111.589} C_DIS
LIN {X 0.176,Y -579.893,Z 1147.412,A 0.000,B 0.000,C 90.000,E1 110.174} C_DIS
LIN {X 0.073,Y -574.222,Z 1147.410,A 0.000,B 0.000,C 90.000,E1 109.704} C_DIS
LIN {X -0.141,Y -568.215,Z 1147.407,A 0.000,B 0.000,C 90.000,E1 109.268} C_DIS
LIN {X 0.038,Y -560.168,Z 1147.404,A 0.000,B 0.000,C 90.000,E1 108.725} C_DIS
LIN {X 0.110,Y -555.466,Z 1147.402,A 0.000,B 0.000,C 90.000,E1 108.417} C_DIS
LIN {X 0.284,Y -551.152,Z 1147.401,A 0.000,B 0.000,C 90.000,E1 108.055} C_DIS
LIN {X 0.226,Y -550.045,Z 1147.400,A 0.000,B 0.000,C 90.000,E1 107.873} C_DIS
LIN {X 0.183,Y -550.020,Z 1147.399,A 0.000,B 0.000,C 90.000,E1 107.873} C_DIS
LIN {X -0.190,Y -549.782,Z 1147.397,A 0.000,B 0.000,C 90.000,E1 107.457} C_DIS
LIN {X 0.127,Y -551.224,Z 1147.385,A 0.000,B 0.000,C 90.000,E1 105.190} C_DIS
LIN {X -0.008,Y -552.859,Z 1147.374,A 0.000,B 0.000,C 90.000,E1 103.244} C_DIS
LIN {X 0.014,Y -554.826,Z 1147.361,A 0.000,B 0.000,C 90.000,E1 101.007} C_DIS
LIN {X 0.275,Y -556.657,Z 1147.350,A 0.000,B 0.000,C 90.000,E1 99.029} C_DIS
LIN {X -0.133,Y -558.302,Z 1147.340,A 0.000,B 0.000,C 90.000,E1 97.125} C_DIS
LIN {X -0.148,Y -559.411,Z 1147.332,A 0.000,B 0.000,C 90.000,E1 95.739} C_DIS
LIN {X -0.203,Y -560.494,Z 1147.324,A 0.000,B 0.000,C 90.000,E1 94.359} C_DIS
LIN {X -0.053,Y -561.982,Z 1147.313,A 0.000,B 0.000,C 90.000,E1 92.407} C_DIS
LIN {X 0.005,Y -563.222,Z 1147.304,A 0.000,B 0.000,C 90.000,E1 90.745} C_DIS
LIN {X -0.031,Y -564.136,Z 1147.297,A 0.000,B 0.000,C 90.000,E1 89.370} C_DIS
LIN {X -0.038,Y -565.020,Z 1147.289,A 0.000,B 0.000,C 90.000,E1 87.993} C_DIS
LIN {X 0.084,Y -565.970,Z 1147.280,A 0.000,B 0.000,C 90.000,E1 86.331} C_DIS
LIN {X 0.251,Y -566.843,Z 1147.271,A 0.000,B 0.000,C 90.000,E1 84.666} C_DIS
LIN {X -0.082,Y -567.700,Z 1147.261,A 0.000,B 0.000,C 90.000,E1 83.053} C_DIS
LIN {X 0.145,Y -568.408,Z 1147.254,A 0.000,B 0.000,C 90.000,E1 81.659} C_DIS
LIN {X 0.121,Y -568.939,Z 1147.248,A 0.000,B 0.000,C 90.000,E1 80.566} C_DIS
LIN {X 0.098,Y -569.743,Z 1147.239,A 0.000,B 0.000,C 90.000,E1 78.926} C_DIS
LIN {X -0.018,Y -570.449,Z 1147.229,A 0.000,B 0.000,C 90.000,E1 77.297} C_DIS
LIN {X 0.124,Y -571.263,Z 1147.220,A 0.000,B 0.000,C 90.000,E1 75.644} C_DIS
LIN {X -0.295,Y -572.448,Z 1147.208,A 0.000,B 0.000,C 90.000,E1 73.504} C_DIS
LIN {X -0.158,Y -573.696,Z 1147.198,A 0.000,B 0.000,C 90.000,E1 71.583} C_DIS
LIN {X 0.189,Y -575.104,Z 1147.187,A 0.000,B 0.000,C 90.000,E1 69.645} C_DIS
LIN {X 0.069,Y -576.563,Z 1147.178,A 0.000,B 0.000,C 90.000,E1 68.028} C_DIS
LIN {X -0.004,Y -578.167,Z 1147.169,A 0.000,B 0.000,C 90.000,E1 66.410} C_DIS
LIN {X -0.339,Y -580.163,Z 1147.157,A 0.000,B 0.000,C 90.000,E1 64.280} C_DIS
LIN {X 0.140,Y -581.615,Z 1147.148,A 0.000,B 0.000,C 90.000,E1 62.615} C_DIS
LIN {X 0.279,Y -583.184,Z 1147.138,A 0.000,B 0.000,C 90.000,E1 60.717} C_DIS
LIN {X -0.087,Y -584.228,Z 1147.130,A 0.000,B 0.000,C 90.000,E1 59.410} C_DIS
LIN {X -0.147,Y -585.117,Z 1147.123,A 0.000,B 0.000,C 90.000,E1 58.074} C_DIS
LIN {X -0.063,Y -585.815,Z 1147.117,A 0.000,B 0.000,C 90.000,E1 56.993} C_DIS
LIN {X -0.134,Y -586.514,Z 1147.111,A 0.000,B 0.000,C 90.000,E1 55.928} C_DIS
LIN {X -0.083,Y -587.769,Z 1147.099,A 0.000,B 0.000,C 90.000,E1 53.783} C_DIS
LIN {X -0.189,Y -588.551,Z 1147.090,A 0.000,B 0.000,C 90.000,E1 52.190} C_DIS
LIN {X 0.150,Y -589.144,Z 1147.084,A 0.000,B 0.000,C 90.000,E1 51.090} C_DIS
LIN {X 0.244,Y -589.635,Z 1147.077,A 0.000,B 0.000,C 90.000,E1 49.747} C_DIS
LIN {X 0.145,Y -589.844,Z 1147.071,A 0.000,B 0.000,C 90.000,E1 48.690} C_DIS
LIN {X 0.044,Y -589.985,Z 1147.065,A 0.000,B 0.000,C 90.000,E1 47.634} C_DIS
LIN {X 0.094,Y -589.879,Z 1147.057,A 0.000,B 0.000,C 90.000,E1 46.296} C_DIS
LIN {X -0.038,Y -589.655,Z 1147.051,A 0.000,B 0.000,C 90.000,E1 45.243} C_DIS
LIN {X -0.171,Y -589.281,Z 1147.045,A 0.000,B 0.000,C 90.000,E1 44.190} C_DIS
LIN {X 0.114,Y -588.657,Z 1147.040,A 0.000,B 0.000,C 90.000,E1 43.095} C_DIS
LIN {X -0.045,Y -587.857,Z 1147.034,A 0.000,B 0.000,C 90.000,E1 42.043} C_DIS
LIN {X -0.178,Y -586.811,Z 1147.028,A 0.000,B 0.000,C 90.000,E1 40.987} C_DIS
LIN {X -0.136,Y -585.250,Z 1147.020,A 0.000,B 0.000,C 90.000,E1 39.644} C_DIS
LIN {X 0.150,Y -583.798,Z 1147.014,A 0.000,B 0.000,C 90.000,E1 38.543} C_DIS
LIN {X -0.047,Y -582.172,Z 1147.008,A 0.000,B 0.000,C 90.000,E1 37.488} C_DIS
LIN {X 0.128,Y -580.695,Z 1147.004,A 0.000,B 0.000,C 90.000,E1 36.664} C_DIS
LIN {X -0.170,Y -578.899,Z 1146.999,A 0.000,B 0.000,C 90.000,E1 35.884} C_DIS
LIN {X 0.319,Y -576.936,Z 1146.995,A 0.000,B 0.000,C 90.000,E1 35.025} C_DIS
LIN {X -0.023,Y -574.646,Z 1146.990,A 0.000,B 0.000,C 90.000,E1 34.246} C_DIS
LIN {X 0.084,Y -572.004,Z 1146.986,A 0.000,B 0.000,C 90.000,E1 33.420} C_DIS
LIN {X 0.035,Y -570.088,Z 1146.983,A 0.000,B 0.000,C 90.000,E1 32.880} C_DIS
LIN {X -0.023,Y -567.964,Z 1146.980,A 0.000,B 0.000,C 90.000,E1 32.339} C_DIS
LIN {X -0.184,Y -563.189,Z 1146.974,A 0.000,B 0.000,C 90.000,E1 31.258} C_DIS
LIN {X -0.013,Y -559.121,Z 1146.969,A 0.000,B 0.000,C 90.000,E1 30.413} C_DIS
LIN {X -0.201,Y -554.002,Z 1146.964,A 0.000,B 0.000,C 90.000,E1 29.461} C_DIS
LIN {X -0.129,Y -549.102,Z 1146.959,A 0.000,B 0.000,C 90.000,E1 28.615} C_DIS
LIN {X 0.014,Y -544.640,Z 1146.955,A 0.000,B 0.000,C 90.000,E1 27.897} C_DIS
LIN {X -0.135,Y -539.891,Z 1146.951,A 0.000,B 0.000,C 90.000,E1 27.206} C_DIS
LIN {X 0.060,Y -535.761,Z 1146.948,A 0.000,B 0.000,C 90.000,E1 26.616} C_DIS
LIN {X -0.061,Y -530.189,Z 1146.944,A 0.000,B 0.000,C 90.000,E1 25.924} C_DIS
LIN {X 0.022,Y -524.390,Z 1146.940,A 0.000,B 0.000,C 90.000,E1 25.207} C_DIS
LIN {X 0.046,Y -516.845,Z 1146.935,A 0.000,B 0.000,C 90.000,E1 24.335} C_DIS
LIN {X 0.122,Y -508.916,Z 1146.930,A 0.000,B 0.000,C 90.000,E1 23.462} C_DIS
LIN {X -0.019,Y -500.622,Z 1146.926,A 0.000,B 0.000,C 90.000,E1 22.642} C_DIS
LIN {X 0.169,Y -496.475,Z 1146.924,A 0.000,B 0.000,C 90.000,E1 22.206} C_DIS
LIN {X 0.058,Y -485.245,Z 1146.918,A 0.000,B 0.000,C 90.000,E1 21.173} C_DIS
LIN {X 0.080,Y -474.996,Z 1146.913,A 0.000,B 0.000,C 90.000,E1 20.248} C_DIS
LIN {X 0.142,Y -466.064,Z 1146.908,A 0.000,B 0.000,C 90.000,E1 19.450} C_DIS
LIN {X 0.069,Y -445.461,Z 1146.898,A 0.000,B 0.000,C 90.000,E1 17.583} C_DIS
LIN {X -0.102,Y -435.249,Z 1146.892,A 0.000,B 0.000,C 90.000,E1 16.622} C_DIS
LIN {X -0.052,Y -419.632,Z 1146.883,A 0.000,B 0.000,C 90.000,E1 14.954} C_DIS
LIN {X -0.041,Y -408.754,Z 1146.876,A 0.000,B 0.000,C 90.000,E1 13.647} C_DIS
LIN {X -0.228,Y -399.851,Z 1146.869,A 0.000,B 0.000,C 90.000,E1 12.479} C_DIS
LIN {X 0.101,Y -395.870,Z 1146.865,A 0.000,B 0.000,C 90.000,E1 11.771} C_DIS
LIN {X -0.008,Y -393.891,Z 1146.863,A 0.000,B 0.000,C 90.000,E1 11.366} C_DIS
LIN {X 0.015,Y -393.232,Z 1146.862,A 0.000,B 0.000,C 90.000,E1 11.186} C_DIS
LIN {X -0.008,Y -392.392,Z 1146.860,A 0.000,B 0.000,C 90.000,E1 10.838} C_DIS
LIN {X -0.037,Y -392.485,Z 1146.857,A 0.000,B 0.000,C 90.000,E1 10.310} C_DIS
LIN {X -0.188,Y -393.667,Z 1146.853,A 0.000,B 0.000,C 90.000,E1 9.613} C_DIS
LIN {X 0.042,Y -397.210,Z 1146.846,A 0.000,B 0.000,C 90.000,E1 8.341} C_DIS
LIN {X -0.046,Y -401.960,Z 1146.839,A 0.000,B 0.000,C 90.000,E1 6.947} C_DIS
LIN {X 0.062,Y -404.796,Z 1146.835,A 0.000,B 0.000,C 90.000,E1 6.258} C_DIS
LIN {X 0.060,Y -406.692,Z 1146.833,A 0.000,B 0.000,C 90.000,E1 5.910} C_DIS
LIN {X 0.042,Y -407.857,Z 1146.832,A 0.000,B 0.000,C 90.000,E1 5.739} C_DIS
LIN {X 0.180,Y -412.323,Z 1146.829,A 0.000,B 0.000,C 90.000,E1 5.220} C_DIS
LIN {X -0.166,Y -417.823,Z 1146.827,A 0.000,B 0.000,C 90.000,E1 4.821} C_DIS
LIN {X -0.023,Y -427.019,Z 1146.823,A 0.000,B 0.000,C 90.000,E1 4.131} C_DIS
LIN {X -0.097,Y -446.545,Z 1146.815,A 0.000,B 0.000,C 90.000,E1 2.751} C_DIS
LIN {X -0.206,Y -461.173,Z 1146.810,A 0.000,B 0.000,C 90.000,E1 1.776} C_DIS
LIN {X 0.205,Y -475.749,Z 1146.804,A 0.000,B 0.000,C 90.000,E1 0.745} C_DIS
LIN {X -0.078,Y -485.150,Z 1146.801,A 0.000,B 0.000,C 90.000,E1 0.115} C_DIS
LIN {X 0.192,Y -492.371,Z 1146.798,A 0.000,B 0.000,C 90.000,E1 359.542} C_DIS
LIN {X 0.088,Y -498.342,Z 1146.795,A 0.000,B 0.000,C 90.000,E1 359.083} C_DIS
LIN {X -0.226,Y -504.206,Z 1146.792,A 0.000,B 0.000,C 90.000,E1 358.625} C_DIS
LIN {X -0.235,Y -509.956,Z 1146.789,A 0.000,B 0.000,C 90.000,E1 358.108} C_DIS
LIN {X -0.052,Y -516.649,Z 1146.786,A 0.000,B 0.000,C 90.000,E1 357.421} C_DIS
LIN {X 0.117,Y -521.931,Z 1146.783,A 0.000,B 0.000,C 90.000,E1 356.846} C_DIS
LIN {X -0.176,Y -528.129,Z 1146.779,A 0.000,B 0.000,C 90.000,E1 356.159} C_DIS
LIN {X -0.201,Y -532.753,Z 1146.775,A 0.000,B 0.000,C 90.000,E1 355.584} C_DIS
LIN {X 0.074,Y -537.833,Z 1146.771,A 0.000,B 0.000,C 90.000,E1 354.837} C_DIS
LIN {X -0.143,Y -542.420,Z 1146.767,A 0.000,B 0.000,C 90.000,E1 354.147} C_DIS
LIN {X -0.061,Y -545.793,Z 1146.764,A 0.000,B 0.000,C 90.000,E1 353.571} C_DIS
LIN {X -0.146,Y -549.565,Z 1146.760,A 0.000,B 0.000,C 90.000,E1 352.875} C_DIS
LIN {X -0.011,Y -552.366,Z 1146.757,A 0.000,B 0.000,C 90.000,E1 352.299} C_DIS
LIN {X -0.034,Y -555.486,Z 1146.753,A 0.000,B 0.000,C 90.000,E1 351.602} C_DIS
LIN {X 0.138,Y -557.861,Z 1146.750,A 0.000,B 0.000,C 90.000,E1 351.027} C_DIS
LIN {X 0.005,Y -561.004,Z 1146.746,A 0.000,B 0.000,C 90.000,E1 350.208} C_DIS
LIN {X -0.191,Y -563.899,Z 1146.741,A 0.000,B 0.000,C 90.000,E1 349.398} C_DIS
LIN {X -0.255,Y -566.508,Z 1146.736,A 0.000,B 0.000,C 90.000,E1 348.578} C_DIS
LIN {X -0.109,Y -569.735,Z 1146.730,A 0.000,B 0.000,C 90.000,E1 347.465} C_DIS
LIN {X 0.079,Y -572.759,Z 1146.724,A 0.000,B 0.000,C 90.000,E1 346.353} C_DIS
LIN {X 0.088,Y -576.289,Z 1146.717,A 0.000,B 0.000,C 90.000,E1 344.991} C_DIS
LIN {X 0.155,Y -579.535,Z 1146.709,A 0.000,B 0.000,C 90.000,E1 343.630} C_DIS
LIN {X 0.223,Y -582.117,Z 1146.703,A 0.000,B 0.000,C 90.000,E1 342.543} C_DIS
LIN {X -0.219,Y -584.542,Z 1146.697,A 0.000,B 0.000,C 90.000,E1 341.511} C_DIS
LIN {X -0.071,Y -586.761,Z 1146.691,A 0.000,B 0.000,C 90.000,E1 340.423} C_DIS
LIN {X 0.099,Y -588.757,Z 1146.685,A 0.000,B 0.000,C 90.000,E1 339.337} C_DIS
LIN {X -0.162,Y -590.908,Z 1146.678,A 0.000,B 0.000,C 90.000,E1 338.028} C_DIS
LIN {X -0.168,Y -591.915,Z 1146.673,A 0.000,B 0.000,C 90.000,E1 337.230} C_DIS
LIN {X 0.067,Y -592.674,Z 1146.669,A 0.000,B 0.000,C 90.000,E1 336.410} C_DIS
LIN {X -0.027,Y -593.482,Z 1146.663,A 0.000,B 0.000,C 90.000,E1 335.357} C_DIS
LIN {X 0.225,Y -593.776,Z 1146.659,A 0.000,B 0.000,C 90.000,E1 334.537} C_DIS
LIN {X -0.056,Y -593.694,Z 1146.654,A 0.000,B 0.000,C 90.000,E1 333.768} C_DIS
LIN {X 0.193,Y -593.279,Z 1146.650,A 0.000,B 0.000,C 90.000,E1 332.948} C_DIS
LIN {X 0.180,Y -592.560,Z 1146.645,A 0.000,B 0.000,C 90.000,E1 332.153} C_DIS
LIN {X -0.216,Y -591.134,Z 1146.640,A 0.000,B 0.000,C 90.000,E1 331.129} C_DIS
LIN {X -0.059,Y -588.879,Z 1146.634,A 0.000,B 0.000,C 90.000,E1 330.049} C_DIS
LIN {X -0.102,Y -586.780,Z 1146.629,A 0.000,B 0.000,C 90.000,E1 329.253} C_DIS
LIN {X -0.168,Y -584.033,Z 1146.625,A 0.000,B 0.000,C 90.000,E1 328.456} C_DIS
LIN {X -0.266,Y -580.635,Z 1146.620,A 0.000,B 0.000,C 90.000,E1 327.661} C_DIS
LIN {X -0.017,Y -577.270,Z 1146.616,A 0.000,B 0.000,C 90.000,E1 326.962} C_DIS
LIN {X -0.114,Y -573.315,Z 1146.613,A 0.000,B 0.000,C 90.000,E1 326.294} C_DIS
LIN {X 0.067,Y -568.847,Z 1146.609,A 0.000,B 0.000,C 90.000,E1 325.595} C_DIS
LIN {X -0.009,Y -564.968,Z 1146.606,A 0.000,B 0.000,C 90.000,E1 325.055} C_DIS
LIN {X -0.004,Y -561.935,Z 1146.604,A 0.000,B 0.000,C 90.000,E1 324.642} C_DIS
LIN {X -0.379,Y -556.112,Z 1146.600,A 0.000,B 0.000,C 90.000,E1 323.989} C_DIS
LIN {X -0.151,Y -548.690,Z 1146.595,A 0.000,B 0.000,C 90.000,E1 323.130} C_DIS
LIN {X -0.257,Y -534.626,Z 1146.587,A 0.000,B 0.000,C 90.000,E1 321.618} C_DIS
LIN {X -0.029,Y -530.938,Z 1146.584,A 0.000,B 0.000,C 90.000,E1 321.170} C_DIS
LIN {X -0.020,Y -528.699,Z 1146.583,A 0.000,B 0.000,C 90.000,E1 320.884} C_DIS
LIN {X 0.277,Y -525.591,Z 1146.580,A 0.000,B 0.000,C 90.000,E1 320.356} C_DIS
LIN {X -0.102,Y -523.470,Z 1146.577,A 0.000,B 0.000,C 90.000,E1 319.908} C_DIS
LIN {X -0.065,Y -522.026,Z 1146.574,A 0.000,B 0.000,C 90.000,E1 319.299} C_DIS
LIN {X 0.121,Y -521.225,Z 1146.569,A 0.000,B 0.000,C 90.000,E1 318.405} C_DIS
LIN {X -0.094,Y -521.083,Z 1146.564,A 0.000,B 0.000,C 90.000,E1 317.553} C_DIS
LIN {X 0.056,Y -521.931,Z 1146.551,A 0.000,B 0.000,C 90.000,E1 315.202} C_DIS
LIN {X -0.005,Y -522.620,Z 1146.542,A 0.000,B 0.000,C 90.000,E1 313.461} C_DIS
LIN {X -0.012,Y -523.276,Z 1146.532,A 0.000,B 0.000,C 90.000,E1 311.714} C_DIS
LIN {X 0.008,Y -524.092,Z 1146.522,A 0.000,B 0.000,C 90.000,E1 309.967} C_DIS
LIN {X 0.029,Y -525.048,Z 1146.512,A 0.000,B 0.000,C 90.000,E1 308.222} C_DIS
LIN {X -0.145,Y -525.942,Z 1146.504,A 0.000,B 0.000,C 90.000,E1 306.790} C_DIS
LIN {X 0.094,Y -527.059,Z 1146.495,A 0.000,B 0.000,C 90.000,E1 305.025} C_DIS
LIN {X 0.088,Y -528.004,Z 1146.487,A 0.000,B 0.000,C 90.000,E1 303.579} C_DIS
LIN {X 0.172,Y -529.532,Z 1146.474,A 0.000,B 0.000,C 90.000,E1 301.258} C_DIS
LIN {X -0.048,Y -530.357,Z 1146.467,A 0.000,B 0.000,C 90.000,E1 300.129} C_DIS
LIN {X -0.090,Y -531.306,Z 1146.459,A 0.000,B 0.000,C 90.000,E1 298.693} C_DIS
LIN {X 0.176,Y -531.882,Z 1146.453,A 0.000,B 0.000,C 90.000,E1 297.513} C_DIS
LIN {X -0.086,Y -532.275,Z 1146.445,A 0.000,B 0.000,C 90.000,E1 296.104} C_DIS
LIN {X -0.058,Y -532.469,Z 1146.439,A 0.000,B 0.000,C 90.000,E1 294.951} C_DIS
LIN {X 0.138,Y -532.507,Z 1146.429,A 0.000,B 0.000,C 90.000,E1 293.206} C_DIS
LIN {X -0.157,Y -532.469,Z 1146.418,A 0.000,B 0.000,C 90.000,E1 291.227} C_DIS
LIN {X -0.054,Y -532.328,Z 1146.411,A 0.000,B 0.000,C 90.000,E1 290.066} C_DIS
LIN {X 0.237,Y -531.985,Z 1146.404,A 0.000,B 0.000,C 90.000,E1 288.598} C_DIS
LIN {X 0.156,Y -531.658,Z 1146.397,A 0.000,B 0.000,C 90.000,E1 287.457} C_DIS
LIN {X 0.101,Y -531.030,Z 1146.389,A 0.000,B 0.000,C 90.000,E1 286.024} C_DIS
LIN {X 0.031,Y -530.373,Z 1146.381,A 0.000,B 0.000,C 90.000,E1 284.592} C_DIS
LIN {X 0.292,Y -529.730,Z 1146.375,A 0.000,B 0.000,C 90.000,E1 283.411} C_DIS
LIN {X -0.027,Y -528.663,Z 1146.365,A 0.000,B 0.000,C 90.000,E1 281.715} C_DIS
LIN {X 0.126,Y -527.850,Z 1146.357,A 0.000,B 0.000,C 90.000,E1 280.254} C_DIS
LIN {X 0.145,Y -527.239,Z 1146.351,A 0.000,B 0.000,C 90.000,E1 279.095} C_DIS
LIN {X 0.145,Y -526.072,Z 1146.339,A 0.000,B 0.000,C 90.000,E1 277.068} C_DIS
LIN {X 0.091,Y -525.148,Z 1146.330,A 0.000,B 0.000,C 90.000,E1 275.334} C_DIS
LIN {X -0.127,Y -524.286,Z 1146.318,A 0.000,B 0.000,C 90.000,E1 273.326} C_DIS
LIN {X 0.198,Y -523.583,Z 1146.309,A 0.000,B 0.000,C 90.000,E1 271.547} C_DIS
LIN {X -0.047,Y -522.862,Z 1146.299,A 0.000,B 0.000,C 90.000,E1 269.828} C_DIS
LIN {X 0.181,Y -521.905,Z 1146.288,A 0.000,B 0.000,C 90.000,E1 267.764} C_DIS
LIN {X -0.093,Y -521.084,Z 1146.278,A 0.000,B 0.000,C 90.000,E1 266.045} C_DIS
LIN {X -0.241,Y -520.378,Z 1146.271,A 0.000,B 0.000,C 90.000,E1 264.894} C_DIS
LIN {X 0.121,Y -519.475,Z 1146.265,A 0.000,B 0.000,C 90.000,E1 263.685} C_DIS
LIN {X -0.088,Y -517.400,Z 1146.254,A 0.000,B 0.000,C 90.000,E1 261.659} C_DIS
LIN {X 0.152,Y -515.304,Z 1146.242,A 0.000,B 0.000,C 90.000,E1 259.577} C_DIS
LIN {X 0.086,Y -513.015,Z 1146.229,A 0.000,B 0.000,C 90.000,E1 257.229} C_DIS
LIN {X -0.009,Y -511.152,Z 1146.218,A 0.000,B 0.000,C 90.000,E1 255.172} C_DIS
LIN {X 0.150,Y -509.566,Z 1146.208,A 0.000,B 0.000,C 90.000,E1 253.378} C_DIS
LIN {X -0.208,Y -507.886,Z 1146.198,A 0.000,B 0.000,C 90.000,E1 251.638} C_DIS
LIN {X 0.014,Y -506.703,Z 1146.191,A 0.000,B 0.000,C 90.000,E1 250.423} C_DIS
LIN {X 0.017,Y -504.537,Z 1146.180,A 0.000,B 0.000,C 90.000,E1 248.337} C_DIS
LIN {X -0.016,Y -502.892,Z 1146.171,A 0.000,B 0.000,C 90.000,E1 246.847} C_DIS
LIN {X -0.159,Y -501.453,Z 1146.165,A 0.000,B 0.000,C 90.000,E1 245.665} C_DIS
LIN {X -0.160,Y -498.615,Z 1146.153,A 0.000,B 0.000,C 90.000,E1 243.563} C_DIS
LIN {X 0.110,Y -496.450,Z 1146.145,A 0.000,B 0.000,C 90.000,E1 242.025} C_DIS
LIN {X -0.138,Y -494.636,Z 1146.138,A 0.000,B 0.000,C 90.000,E1 240.845} C_DIS
LIN {X 0.011,Y -492.769,Z 1146.131,A 0.000,B 0.000,C 90.000,E1 239.616} C_DIS
LIN {X 0.041,Y -489.912,Z 1146.121,A 0.000,B 0.000,C 90.000,E1 237.788} C_DIS
LIN {X -0.163,Y -486.511,Z 1146.109,A 0.000,B 0.000,C 90.000,E1 235.674} C_DIS
LIN {X 0.085,Y -483.065,Z 1146.097,A 0.000,B 0.000,C 90.000,E1 233.497} C_DIS
LIN {X 0.030,Y -480.994,Z 1146.090,A 0.000,B 0.000,C 90.000,E1 232.271} C_DIS
LIN {X -0.149,Y -477.917,Z 1146.080,A 0.000,B 0.000,C 90.000,E1 230.436} C_DIS
LIN {X 0.116,Y -475.255,Z 1146.072,A 0.000,B 0.000,C 90.000,E1 228.852} C_DIS
LIN {X 0.066,Y -472.087,Z 1146.061,A 0.000,B 0.000,C 90.000,E1 226.986} C_DIS
LIN {X -0.191,Y -465.727,Z 1146.038,A 0.000,B 0.000,C 90.000,E1 222.933} C_DIS
LIN {X 0.205,Y -463.534,Z 1146.028,A 0.000,B 0.000,C 90.000,E1 220.987} C_DIS
LIN {X 0.042,Y -461.274,Z 1146.016,A 0.000,B 0.000,C 90.000,E1 218.785} C_DIS
LIN {X -0.174,Y -459.367,Z 1146.003,A 0.000,B 0.000,C 90.000,E1 216.583} C_DIS
LIN {X -0.233,Y -456.211,Z 1145.966,A 0.000,B 0.000,C 90.000,E1 209.873} C_DIS
LIN {X 0.184,Y -456.519,Z 1145.955,A 0.000,B 0.000,C 90.000,E1 207.897} C_DIS
LIN {X 0.188,Y -458.136,Z 1145.941,A 0.000,B 0.000,C 90.000,E1 205.335} C_DIS
LIN {X -0.056,Y -460.970,Z 1145.928,A 0.000,B 0.000,C 90.000,E1 203.131} C_DIS
LIN {X -0.215,Y -465.649,Z 1145.914,A 0.000,B 0.000,C 90.000,E1 200.610} C_DIS
LIN {X 0.160,Y -470.110,Z 1145.904,A 0.000,B 0.000,C 90.000,E1 198.671} C_DIS
LIN {X 0.016,Y -476.288,Z 1145.892,A 0.000,B 0.000,C 90.000,E1 196.496} C_DIS
LIN {X 0.087,Y -484.555,Z 1145.878,A 0.000,B 0.000,C 90.000,E1 194.008} C_DIS
LIN {X -0.068,Y -490.982,Z 1145.868,A 0.000,B 0.000,C 90.000,E1 192.187} C_DIS
LIN {X -0.087,Y -497.670,Z 1145.858,A 0.000,B 0.000,C 90.000,E1 190.366} C_DIS
LIN {X -0.144,Y -504.449,Z 1145.848,A 0.000,B 0.000,C 90.000,E1 188.568} C_DIS
LIN {X -0.071,Y -510.231,Z 1145.839,A 0.000,B 0.000,C 90.000,E1 187.068} C_DIS
LIN {X 0.118,Y -515.913,Z 1145.831,A 0.000,B 0.000,C 90.000,E1 185.568} C_DIS
LIN {X -0.174,Y -522.678,Z 1145.821,A 0.000,B 0.000,C 90.000,E1 183.841} C_DIS
LIN {X 0.196,Y -527.181,Z 1145.815,A 0.000,B 0.000,C 90.000,E1 182.636} C_DIS
LIN {X 0.080,Y -533.889,Z 1145.805,A 0.000,B 0.000,C 90.000,E1 180.917} C_DIS
LIN {X 0.087,Y -539.495,Z 1145.797,A 0.000,B 0.000,C 90.000,E1 179.484} C_DIS
LIN {X -0.267,Y -547.330,Z 1145.786,A 0.000,B 0.000,C 90.000,E1 177.535} C_DIS
LIN {X 0.087,Y -554.026,Z 1145.777,A 0.000,B 0.000,C 90.000,E1 175.812} C_DIS
LIN {X -0.043,Y -559.660,Z 1145.769,A 0.000,B 0.000,C 90.000,E1 174.432} C_DIS
LIN {X 0.073,Y -566.318,Z 1145.760,A 0.000,B 0.000,C 90.000,E1 172.761} C_DIS
LIN {X -0.164,Y -572.938,Z 1145.751,A 0.000,B 0.000,C 90.000,E1 171.141} C_DIS
LIN {X 0.180,Y -578.377,Z 1145.743,A 0.000,B 0.000,C 90.000,E1 169.746} C_DIS
LIN {X -0.052,Y -585.778,Z 1145.733,A 0.000,B 0.000,C 90.000,E1 167.881} C_DIS
LIN {X 0.053,Y -590.859,Z 1145.725,A 0.000,B 0.000,C 90.000,E1 166.533} C_DIS
LIN {X 0.111,Y -594.787,Z 1145.719,A 0.000,B 0.000,C 90.000,E1 165.463} C_DIS
LIN {X -0.058,Y -599.387,Z 1145.712,A 0.000,B 0.000,C 90.000,E1 164.157} C_DIS
LIN {X 0.020,Y -603.765,Z 1145.705,A 0.000,B 0.000,C 90.000,E1 162.834} C_DIS
LIN {X 0.259,Y -607.120,Z 1145.699,A 0.000,B 0.000,C 90.000,E1 161.764} C_DIS
LIN {X 0.152,Y -610.347,Z 1145.693,A 0.000,B 0.000,C 90.000,E1 160.732} C_DIS
LIN {X 0.043,Y -614.161,Z 1145.686,A 0.000,B 0.000,C 90.000,E1 159.444} C_DIS
LIN {X 0.001,Y -617.694,Z 1145.679,A 0.000,B 0.000,C 90.000,E1 158.156} C_DIS
LIN {X 0.007,Y -621.203,Z 1145.672,A 0.000,B 0.000,C 90.000,E1 156.869} C_DIS
LIN {X -0.251,Y -625.837,Z 1145.662,A 0.000,B 0.000,C 90.000,E1 155.101} C_DIS
LIN {X -0.191,Y -628.425,Z 1145.656,A 0.000,B 0.000,C 90.000,E1 154.076} C_DIS
LIN {X -0.062,Y -631.481,Z 1145.649,A 0.000,B 0.000,C 90.000,E1 152.794} C_DIS
LIN {X 0.112,Y -634.382,Z 1145.642,A 0.000,B 0.000,C 90.000,E1 151.513} C_DIS
LIN {X 0.079,Y -637.157,Z 1145.635,A 0.000,B 0.000,C 90.000,E1 150.255} C_DIS
LIN {X 0.144,Y -640.262,Z 1145.626,A 0.000,B 0.000,C 90.000,E1 148.742} C_DIS
LIN {X -0.002,Y -642.734,Z 1145.620,A 0.000,B 0.000,C 90.000,E1 147.502} C_DIS
LIN {X -0.043,Y -645.476,Z 1145.611,A 0.000,B 0.000,C 90.000,E1 146.008} C_DIS
LIN {X 0.323,Y -648.056,Z 1145.603,A 0.000,B 0.000,C 90.000,E1 144.482} C_DIS
LIN {X 0.205,Y -650.548,Z 1145.595,A 0.000,B 0.000,C 90.000,E1 143.004} C_DIS
LIN {X -0.070,Y -654.365,Z 1145.582,A 0.000,B 0.000,C 90.000,E1 140.803} C_DIS
LIN {X -0.237,Y -657.662,Z 1145.573,A 0.000,B 0.000,C 90.000,E1 139.094} C_DIS
LIN {X -0.395,Y -661.123,Z 1145.563,A 0.000,B 0.000,C 90.000,E1 137.391} C_DIS
LIN {X -0.025,Y -665.016,Z 1145.552,A 0.000,B 0.000,C 90.000,E1 135.405} C_DIS
LIN {X -0.020,Y -669.837,Z 1145.540,A 0.000,B 0.000,C 90.000,E1 133.218} C_DIS
LIN {X -0.328,Y -674.415,Z 1145.529,A 0.000,B 0.000,C 90.000,E1 131.310} C_DIS
LIN {X 0.005,Y -679.082,Z 1145.519,A 0.000,B 0.000,C 90.000,E1 129.358} C_DIS
LIN {X -0.180,Y -682.165,Z 1145.512,A 0.000,B 0.000,C 90.000,E1 128.177} C_DIS
LIN {X -0.129,Y -686.366,Z 1145.503,A 0.000,B 0.000,C 90.000,E1 126.503} C_DIS
LIN {X -0.073,Y -689.347,Z 1145.496,A 0.000,B 0.000,C 90.000,E1 125.311} C_DIS
LIN {X -0.325,Y -692.826,Z 1145.488,A 0.000,B 0.000,C 90.000,E1 123.913} C_DIS
LIN {X 0.032,Y -695.541,Z 1145.482,A 0.000,B 0.000,C 90.000,E1 122.704} C_DIS
LIN {X 0.197,Y -697.622,Z 1145.477,A 0.000,B 0.000,C 90.000,E1 121.750} C_DIS
LIN {X 0.125,Y -698.970,Z 1145.473,A 0.000,B 0.000,C 90.000,E1 121.052} C_DIS
LIN {X 0.228,Y -700.993,Z 1145.466,A 0.000,B 0.000,C 90.000,E1 119.873} C_DIS
LIN {X 0.035,Y -703.520,Z 1145.458,A 0.000,B 0.000,C 90.000,E1 118.487} C_DIS
LIN {X 0.262,Y -704.613,Z 1145.454,A 0.000,B 0.000,C 90.000,E1 117.769} C_DIS
LIN {X -0.115,Y -705.221,Z 1145.452,A 0.000,B 0.000,C 90.000,E1 117.334} C_DIS
LIN {X -0.163,Y -705.703,Z 1145.449,A 0.000,B 0.000,C 90.000,E1 116.873} C_DIS
LIN {X 0.061,Y -706.225,Z 1145.444,A 0.000,B 0.000,C 90.000,E1 115.924} C_DIS
LIN {X 0.304,Y -706.436,Z 1145.440,A 0.000,B 0.000,C 90.000,E1 115.207} C_DIS
LIN {X 0.242,Y -706.264,Z 1145.436,A 0.000,B 0.000,C 90.000,E1 114.515} C_DIS
LIN {X -0.110,Y -705.400,Z 1145.434,A 0.000,B 0.000,C 90.000,E1 114.079} C_DIS
LIN {X 0.179,Y -704.777,Z 1145.432,A 0.000,B 0.000,C 90.000,E1 113.823} C_DIS
LIN {X -0.180,Y -702.803,Z 1145.430,A 0.000,B 0.000,C 90.000,E1 113.387} C_DIS
LIN {X -0.040,Y -702.152,Z 1145.429,A 0.000,B 0.000,C 90.000,E1 113.259} C_DIS
LIN {X 0.098,Y -701.174,Z 1145.429,A 0.000,B 0.000,C 90.000,E1 113.131} C_DIS
LIN {X 0.372,Y -696.476,Z 1145.426,A 0.000,B 0.000,C 90.000,E1 112.642} C_DIS
LIN {X -0.375,Y -694.656,Z 1145.425,A 0.000,B 0.000,C 90.000,E1 112.589} C_DIS
LIN {X -0.254,Y -686.285,Z 1145.424,A 0.000,B 0.000,C 90.000,E1 112.280} C_DIS
LIN {X -0.069,Y -682.590,Z 1145.423,A 0.000,B 0.000,C 90.000,E1 112.206} C_DIS
LIN {X -0.070,Y -676.459,Z 1145.423,A 0.000,B 0.000,C 90.000,E1 112.153} C_DIS
LIN {X -0.117,Y -603.403,Z 1145.423,A 0.000,B 0.000,C 90.000,E1 112.153} C_DIS
LIN {X -0.108,Y -600.325,Z 1145.422,A 0.000,B 0.000,C 90.000,E1 111.950} C_DIS
LIN {X 0.125,Y -594.404,Z 1145.419,A 0.000,B 0.000,C 90.000,E1 111.461} C_DIS
LIN {X 0.058,Y -579.756,Z 1145.412,A 0.000,B 0.000,C 90.000,E1 110.174} C_DIS
LIN {X -0.038,Y -574.078,Z 1145.410,A 0.000,B 0.000,C 90.000,E1 109.704} C_DIS
LIN {X -0.253,Y -568.087,Z 1145.407,A 0.000,B 0.000,C 90.000,E1 109.268} C_DIS
LIN {X -0.054,Y -559.997,Z 1145.404,A 0.000,B 0.000,C 90.000,E1 108.725} C_DIS
LIN {X 0.129,Y -555.450,Z 1145.402,A 0.000,B 0.000,C 90.000,E1 108.417} C_DIS
LIN {X 0.307,Y -551.104,Z 1145.401,A 0.000,B 0.000,C 90.000,E1 108.055} C_DIS
LIN {X 0.222,Y -549.972,Z 1145.400,A 0.000,B 0.000,C 90.000,E1 107.873} C_DIS
LIN {X 0.182,Y -549.959,Z 1145.399,A 0.000,B 0.000,C 90.000,E1 107.873} C_DIS
LIN {X -0.020,Y -549.716,Z 1145.397,A 0.000,B 0.000,C 90.000,E1 107.457} C_DIS
LIN {X -0.237,Y -551.154,Z 1145.385,A 0.000,B 0.000,C 90.000,E1 105.245} C_DIS
LIN {X 0.158,Y -552.754,Z 1145.374,A 0.000,B 0.000,C 90.000,E1 103.244} C_DIS
LIN {X 0.053,Y -554.461,Z 1145.363,A 0.000,B 0.000,C 90.000,E1 101.299} C_DIS
LIN {X -0.200,Y -556.549,Z 1145.350,A 0.000,B 0.000,C 90.000,E1 99.095} C_DIS
LIN {X 0.028,Y -558.195,Z 1145.340,A 0.000,B 0.000,C 90.000,E1 97.125} C_DIS
LIN {X 0.011,Y -559.338,Z 1145.332,A 0.000,B 0.000,C 90.000,E1 95.739} C_DIS
LIN {X 0.042,Y -560.635,Z 1145.323,A 0.000,B 0.000,C 90.000,E1 94.073} C_DIS
LIN {X 0.104,Y -561.938,Z 1145.313,A 0.000,B 0.000,C 90.000,E1 92.407} C_DIS
LIN {X 0.161,Y -563.149,Z 1145.304,A 0.000,B 0.000,C 90.000,E1 90.745} C_DIS
LIN {X 0.124,Y -564.049,Z 1145.297,A 0.000,B 0.000,C 90.000,E1 89.370} C_DIS
LIN {X 0.116,Y -564.945,Z 1145.289,A 0.000,B 0.000,C 90.000,E1 87.993} C_DIS
LIN {X 0.235,Y -565.870,Z 1145.280,A 0.000,B 0.000,C 90.000,E1 86.331} C_DIS
LIN {X -0.270,Y -566.609,Z 1145.272,A 0.000,B 0.000,C 90.000,E1 85.008} C_DIS
LIN {X -0.033,Y -567.444,Z 1145.263,A 0.000,B 0.000,C 90.000,E1 83.337} C_DIS
LIN {X 0.291,Y -568.272,Z 1145.254,A 0.000,B 0.000,C 90.000,E1 81.659} C_DIS
LIN {X -0.117,Y -568.921,Z 1145.246,A 0.000,B 0.000,C 90.000,E1 80.330} C_DIS
LIN {X 0.239,Y -569.575,Z 1145.239,A 0.000,B 0.000,C 90.000,E1 78.926} C_DIS
LIN {X 0.121,Y -570.324,Z 1145.229,A 0.000,B 0.000,C 90.000,E1 77.297} C_DIS
LIN {X -0.108,Y -571.247,Z 1145.219,A 0.000,B 0.000,C 90.000,E1 75.408} C_DIS
LIN {X 0.182,Y -572.475,Z 1145.207,A 0.000,B 0.000,C 90.000,E1 73.196} C_DIS
LIN {X -0.213,Y -573.754,Z 1145.196,A 0.000,B 0.000,C 90.000,E1 71.329} C_DIS
LIN {X -0.224,Y -574.991,Z 1145.187,A 0.000,B 0.000,C 90.000,E1 69.699} C_DIS
LIN {X 0.193,Y -576.449,Z 1145.178,A 0.000,B 0.000,C 90.000,E1 68.028} C_DIS
LIN {X -0.114,Y -578.048,Z 1145.169,A 0.000,B 0.000,C 90.000,E1 66.433} C_DIS
LIN {X -0.220,Y -580.029,Z 1145.157,A 0.000,B 0.000,C 90.000,E1 64.280} C_DIS
LIN {X 0.256,Y -581.480,Z 1145.148,A 0.000,B 0.000,C 90.000,E1 62.615} C_DIS
LIN {X -0.269,Y -582.825,Z 1145.139,A 0.000,B 0.000,C 90.000,E1 61.051} C_DIS
LIN {X 0.155,Y -583.863,Z 1145.132,A 0.000,B 0.000,C 90.000,E1 59.665} C_DIS
LIN {X 0.094,Y -584.790,Z 1145.124,A 0.000,B 0.000,C 90.000,E1 58.329} C_DIS
LIN {X 0.042,Y -585.632,Z 1145.117,A 0.000,B 0.000,C 90.000,E1 56.993} C_DIS
LIN {X -0.173,Y -586.445,Z 1145.109,A 0.000,B 0.000,C 90.000,E1 55.674} C_DIS
LIN {X 0.014,Y -587.576,Z 1145.099,A 0.000,B 0.000,C 90.000,E1 53.783} C_DIS
LIN {X 0.103,Y -588.495,Z 1145.089,A 0.000,B 0.000,C 90.000,E1 51.904} C_DIS
LIN {X -0.017,Y -589.047,Z 1145.083,A 0.000,B 0.000,C 90.000,E1 50.848} C_DIS
LIN {X -0.302,Y -589.497,Z 1145.075,A 0.000,B 0.000,C 90.000,E1 49.542} C_DIS
LIN {X -0.069,Y -589.673,Z 1145.066,A 0.000,B 0.000,C 90.000,E1 47.919} C_DIS
LIN {X -0.016,Y -589.615,Z 1145.059,A 0.000,B 0.000,C 90.000,E1 46.581} C_DIS
LIN {X -0.316,Y -589.507,Z 1145.054,A 0.000,B 0.000,C 90.000,E1 45.810} C_DIS
LIN {X -0.037,Y -589.169,Z 1145.048,A 0.000,B 0.000,C 90.000,E1 44.717} C_DIS
LIN {X -0.348,Y -588.801,Z 1145.044,A 0.000,B 0.000,C 90.000,E1 43.947} C_DIS
LIN {X -0.070,Y -588.169,Z 1145.038,A 0.000,B 0.000,C 90.000,E1 42.852} C_DIS
LIN {X 0.198,Y -587.292,Z 1145.032,A 0.000,B 0.000,C 90.000,E1 41.757} C_DIS
LIN {X 0.061,Y -586.144,Z 1145.026,A 0.000,B 0.000,C 90.000,E1 40.701} C_DIS
LIN {X -0.090,Y -584.891,Z 1145.020,A 0.000,B 0.000,C 90.000,E1 39.644} C_DIS
LIN {X 0.192,Y -583.425,Z 1145.014,A 0.000,B 0.000,C 90.000,E1 38.543} C_DIS
LIN {X -0.365,Y -581.775,Z 1145.008,A 0.000,B 0.000,C 90.000,E1 37.523} C_DIS
LIN {X 0.160,Y -580.291,Z 1145.004,A 0.000,B 0.000,C 90.000,E1 36.664} C_DIS
LIN {X -0.143,Y -578.474,Z 1144.999,A 0.000,B 0.000,C 90.000,E1 35.884} C_DIS
LIN {X -0.306,Y -575.757,Z 1144.993,A 0.000,B 0.000,C 90.000,E1 34.818} C_DIS
LIN {X -0.005,Y -574.161,Z 1144.990,A 0.000,B 0.000,C 90.000,E1 34.246} C_DIS
LIN {X 0.096,Y -571.462,Z 1144.986,A 0.000,B 0.000,C 90.000,E1 33.420} C_DIS
LIN {X 0.045,Y -569.550,Z 1144.983,A 0.000,B 0.000,C 90.000,E1 32.880} C_DIS
LIN {X -0.018,Y -567.408,Z 1144.980,A 0.000,B 0.000,C 90.000,E1 32.339} C_DIS
LIN {X -0.186,Y -562.594,Z 1144.974,A 0.000,B 0.000,C 90.000,E1 31.258} C_DIS
LIN {X -0.022,Y -558.464,Z 1144.969,A 0.000,B 0.000,C 90.000,E1 30.413} C_DIS
LIN {X 0.264,Y -553.316,Z 1144.964,A 0.000,B 0.000,C 90.000,E1 29.411} C_DIS
LIN {X -0.035,Y -549.241,Z 1144.960,A 0.000,B 0.000,C 90.000,E1 28.743} C_DIS
LIN {X -0.015,Y -543.948,Z 1144.955,A 0.000,B 0.000,C 90.000,E1 27.897} C_DIS
LIN {X 0.076,Y -539.156,Z 1144.951,A 0.000,B 0.000,C 90.000,E1 27.180} C_DIS
LIN {X -0.118,Y -533.842,Z 1144.947,A 0.000,B 0.000,C 90.000,E1 26.488} C_DIS
LIN {X 0.116,Y -525.849,Z 1144.942,A 0.000,B 0.000,C 90.000,E1 25.463} C_DIS
LIN {X -0.028,Y -520.927,Z 1144.938,A 0.000,B 0.000,C 90.000,E1 24.899} C_DIS
LIN {X 0.154,Y -514.425,Z 1144.934,A 0.000,B 0.000,C 90.000,E1 24.155} C_DIS
LIN {X 0.099,Y -508.050,Z 1144.930,A 0.000,B 0.000,C 90.000,E1 23.462} C_DIS
LIN {X -0.124,Y -497.132,Z 1144.924,A 0.000,B 0.000,C 90.000,E1 22.386} C_DIS
LIN {X 0.182,Y -485.638,Z 1144.918,A 0.000,B 0.000,C 90.000,E1 21.280} C_DIS
LIN {X 0.153,Y -474.124,Z 1144.913,A 0.000,B 0.000,C 90.000,E1 20.248} C_DIS
LIN {X 0.047,Y -467.023,Z 1144.909,A 0.000,B 0.000,C 90.000,E1 19.631} C_DIS
LIN {X 0.175,Y -445.278,Z 1144.898,A 0.000,B 0.000,C 90.000,E1 17.638} C_DIS
LIN {X 0.200,Y -435.315,Z 1144.893,A 0.000,B 0.000,C 90.000,E1 16.677} C_DIS
LIN {X -0.139,Y -419.732,Z 1144.884,A 0.000,B 0.000,C 90.000,E1 15.064} C_DIS
LIN {X -0.217,Y -408.842,Z 1144.876,A 0.000,B 0.000,C 90.000,E1 13.772} C_DIS
LIN {X -0.017,Y -399.825,Z 1144.870,A 0.000,B 0.000,C 90.000,E1 12.535} C_DIS
LIN {X 0.128,Y -396.042,Z 1144.866,A 0.000,B 0.000,C 90.000,E1 11.895} C_DIS
LIN {X 0.046,Y -393.604,Z 1144.863,A 0.000,B 0.000,C 90.000,E1 11.366} C_DIS
LIN {X 0.086,Y -392.721,Z 1144.861,A 0.000,B 0.000,C 90.000,E1 11.007} C_DIS
LIN {X 0.028,Y -392.351,Z 1144.860,A 0.000,B 0.000,C 90.000,E1 10.838} C_DIS
LIN {X -0.001,Y -392.504,Z 1144.857,A 0.000,B 0.000,C 90.000,E1 10.310} C_DIS
LIN {X -0.152,Y -393.772,Z 1144.853,A 0.000,B 0.000,C 90.000,E1 9.613} C_DIS
LIN {X -0.005,Y -397.990,Z 1144.845,A 0.000,B 0.000,C 90.000,E1 8.106} C_DIS
LIN {X -0.137,Y -402.837,Z 1144.837,A 0.000,B 0.000,C 90.000,E1 6.720} C_DIS
LIN {X -0.169,Y -405.028,Z 1144.834,A 0.000,B 0.000,C 90.000,E1 6.201} C_DIS
LIN {X -0.058,Y -407.208,Z 1144.832,A 0.000,B 0.000,C 90.000,E1 5.796} C_DIS
LIN {X -0.021,Y -411.422,Z 1144.829,A 0.000,B 0.000,C 90.000,E1 5.277} C_DIS
LIN {X -0.157,Y -417.083,Z 1144.827,A 0.000,B 0.000,C 90.000,E1 4.821} C_DIS
LIN {X 0.111,Y -425.305,Z 1144.823,A 0.000,B 0.000,C 90.000,E1 4.188} C_DIS
LIN {X -0.002,Y -444.831,Z 1144.816,A 0.000,B 0.000,C 90.000,E1 2.808} C_DIS
LIN {X -0.135,Y -459.499,Z 1144.810,A 0.000,B 0.000,C 90.000,E1 1.835} C_DIS
LIN {X -0.187,Y -472.399,Z 1144.805,A 0.000,B 0.000,C 90.000,E1 0.974} C_DIS
LIN {X 0.145,Y -478.559,Z 1144.803,A 0.000,B 0.000,C 90.000,E1 0.516} C_DIS
LIN {X -0.051,Y -484.577,Z 1144.801,A 0.000,B 0.000,C 90.000,E1 0.115} C_DIS
LIN {X -0.233,Y -491.811,Z 1144.798,A 0.000,B 0.000,C 90.000,E1 359.599} C_DIS
LIN {X 0.151,Y -497.839,Z 1144.795,A 0.000,B 0.000,C 90.000,E1 359.083} C_DIS
LIN {X -0.161,Y -503.788,Z 1144.792,A 0.000,B 0.000,C 90.000,E1 358.625} C_DIS
LIN {X -0.025,Y -510.635,Z 1144.789,A 0.000,B 0.000,C 90.000,E1 357.993} C_DIS
LIN {X 0.141,Y -517.352,Z 1144.785,A 0.000,B 0.000,C 90.000,E1 357.306} C_DIS
LIN {X -0.006,Y -522.433,Z 1144.782,A 0.000,B 0.000,C 90.000,E1 356.788} C_DIS
LIN {X -0.069,Y -527.513,Z 1144.779,A 0.000,B 0.000,C 90.000,E1 356.216} C_DIS
LIN {X 0.194,Y -533.247,Z 1144.775,A 0.000,B 0.000,C 90.000,E1 355.469} C_DIS
LIN {X 0.247,Y -537.377,Z 1144.772,A 0.000,B 0.000,C 90.000,E1 354.894} C_DIS
LIN {X 0.028,Y -542.028,Z 1144.768,A 0.000,B 0.000,C 90.000,E1 354.204} C_DIS
LIN {X 0.108,Y -545.487,Z 1144.765,A 0.000,B 0.000,C 90.000,E1 353.628} C_DIS
LIN {X 0.022,Y -549.361,Z 1144.761,A 0.000,B 0.000,C 90.000,E1 352.932} C_DIS
LIN {X -0.100,Y -552.810,Z 1144.757,A 0.000,B 0.000,C 90.000,E1 352.243} C_DIS
LIN {X 0.134,Y -555.376,Z 1144.754,A 0.000,B 0.000,C 90.000,E1 351.659} C_DIS
LIN {X -0.244,Y -557.779,Z 1144.751,A 0.000,B 0.000,C 90.000,E1 351.141} C_DIS
LIN {X 0.082,Y -560.972,Z 1144.746,A 0.000,B 0.000,C 90.000,E1 350.274} C_DIS
LIN {X -0.017,Y -563.912,Z 1144.741,A 0.000,B 0.000,C 90.000,E1 349.454} C_DIS
LIN {X 0.093,Y -567.385,Z 1144.735,A 0.000,B 0.000,C 90.000,E1 348.342} C_DIS
LIN {X 0.255,Y -570.590,Z 1144.729,A 0.000,B 0.000,C 90.000,E1 347.229} C_DIS
LIN {X -0.099,Y -573.611,Z 1144.723,A 0.000,B 0.000,C 90.000,E1 346.172} C_DIS
LIN {X 0.281,Y -576.487,Z 1144.717,A 0.000,B 0.000,C 90.000,E1 345.046} C_DIS
LIN {X 0.009,Y -580.446,Z 1144.708,A 0.000,B 0.000,C 90.000,E1 343.449} C_DIS
LIN {X -0.248,Y -583.643,Z 1144.701,A 0.000,B 0.000,C 90.000,E1 342.127} C_DIS
LIN {X 0.292,Y -586.518,Z 1144.693,A 0.000,B 0.000,C 90.000,E1 340.732} C_DIS
LIN {X 0.241,Y -588.098,Z 1144.689,A 0.000,B 0.000,C 90.000,E1 339.934} C_DIS
LIN {X -0.122,Y -590.020,Z 1144.683,A 0.000,B 0.000,C 90.000,E1 338.901} C_DIS
LIN {X -0.249,Y -591.720,Z 1144.677,A 0.000,B 0.000,C 90.000,E1 337.847} C_DIS
LIN {X 0.092,Y -593.168,Z 1144.669,A 0.000,B 0.000,C 90.000,E1 336.485} C_DIS
LIN {X 0.246,Y -594.014,Z 1144.664,A 0.000,B 0.000,C 90.000,E1 335.409} C_DIS
LIN {X -0.285,Y -594.403,Z 1144.659,A 0.000,B 0.000,C 90.000,E1 334.665} C_DIS
LIN {X -0.027,Y -594.349,Z 1144.655,A 0.000,B 0.000,C 90.000,E1 333.845} C_DIS
LIN {X -0.034,Y -594.013,Z 1144.650,A 0.000,B 0.000,C 90.000,E1 333.050} C_DIS
LIN {X -0.217,Y -593.639,Z 1144.647,A 0.000,B 0.000,C 90.000,E1 332.538} C_DIS
LIN {X 0.025,Y -592.742,Z 1144.643,A 0.000,B 0.000,C 90.000,E1 331.719} C_DIS
LIN {X 0.013,Y -591.615,Z 1144.639,A 0.000,B 0.000,C 90.000,E1 330.923} C_DIS
LIN {X -0.007,Y -589.919,Z 1144.634,A 0.000,B 0.000,C 90.000,E1 330.127} C_DIS
LIN {X -0.042,Y -587.902,Z 1144.630,A 0.000,B 0.000,C 90.000,E1 329.331} C_DIS
LIN {X -0.159,Y -587.129,Z 1144.628,A 0.000,B 0.000,C 90.000,E1 329.076} C_DIS
LIN {X 0.079,Y -584.275,Z 1144.624,A 0.000,B 0.000,C 90.000,E1 328.250} C_DIS
LIN {X 0.052,Y -581.452,Z 1144.620,A 0.000,B 0.000,C 90.000,E1 327.582} C_DIS
LIN {X -0.006,Y -578.116,Z 1144.616,A 0.000,B 0.000,C 90.000,E1 326.914} C_DIS
LIN {X 0.218,Y -574.227,Z 1144.612,A 0.000,B 0.000,C 90.000,E1 326.215} C_DIS
LIN {X 0.087,Y -569.858,Z 1144.609,A 0.000,B 0.000,C 90.000,E1 325.548} C_DIS
LIN {X -0.006,Y -564.025,Z 1144.604,A 0.000,B 0.000,C 90.000,E1 324.736} C_DIS
LIN {X -0.004,Y -560.768,Z 1144.602,A 0.000,B 0.000,C 90.000,E1 324.322} C_DIS
LIN {X 0.146,Y -557.491,Z 1144.600,A 0.000,B 0.000,C 90.000,E1 323.909} C_DIS
LIN {X 0.080,Y -550.111,Z 1144.595,A 0.000,B 0.000,C 90.000,E1 323.084} C_DIS
LIN {X 0.072,Y -541.205,Z 1144.590,A 0.000,B 0.000,C 90.000,E1 322.110} C_DIS
LIN {X -0.296,Y -532.283,Z 1144.584,A 0.000,B 0.000,C 90.000,E1 321.170} C_DIS
LIN {X -0.231,Y -529.437,Z 1144.582,A 0.000,B 0.000,C 90.000,E1 320.803} C_DIS
LIN {X 0.183,Y -526.327,Z 1144.579,A 0.000,B 0.000,C 90.000,E1 320.275} C_DIS
LIN {X 0.038,Y -523.681,Z 1144.576,A 0.000,B 0.000,C 90.000,E1 319.666} C_DIS
LIN {X -0.160,Y -522.568,Z 1144.573,A 0.000,B 0.000,C 90.000,E1 319.218} C_DIS
LIN {X 0.098,Y -521.859,Z 1144.570,A 0.000,B 0.000,C 90.000,E1 318.609} C_DIS
LIN {X 0.044,Y -521.610,Z 1144.568,A 0.000,B 0.000,C 90.000,E1 318.324} C_DIS
LIN {X 0.127,Y -521.498,Z 1144.562,A 0.000,B 0.000,C 90.000,E1 317.148} C_DIS
LIN {X 0.209,Y -521.850,Z 1144.556,A 0.000,B 0.000,C 90.000,E1 315.972} C_DIS
LIN {X 0.221,Y -522.451,Z 1144.547,A 0.000,B 0.000,C 90.000,E1 314.514} C_DIS
LIN {X 0.180,Y -523.094,Z 1144.538,A 0.000,B 0.000,C 90.000,E1 312.771} C_DIS
LIN {X 0.045,Y -524.033,Z 1144.525,A 0.000,B 0.000,C 90.000,E1 310.458} C_DIS
LIN {X -0.018,Y -525.300,Z 1144.512,A 0.000,B 0.000,C 90.000,E1 308.141} C_DIS
LIN {X 0.201,Y -526.344,Z 1144.502,A 0.000,B 0.000,C 90.000,E1 306.377} C_DIS
LIN {X 0.021,Y -527.495,Z 1144.493,A 0.000,B 0.000,C 90.000,E1 304.659} C_DIS
LIN {X 0.016,Y -528.414,Z 1144.485,A 0.000,B 0.000,C 90.000,E1 303.214} C_DIS
LIN {X -0.144,Y -529.801,Z 1144.473,A 0.000,B 0.000,C 90.000,E1 301.209} C_DIS
LIN {X 0.071,Y -530.834,Z 1144.465,A 0.000,B 0.000,C 90.000,E1 299.745} C_DIS
LIN {X 0.001,Y -531.923,Z 1144.456,A 0.000,B 0.000,C 90.000,E1 298.025} C_DIS
LIN {X -0.264,Y -532.440,Z 1144.448,A 0.000,B 0.000,C 90.000,E1 296.616} C_DIS
LIN {X 0.156,Y -532.725,Z 1144.438,A 0.000,B 0.000,C 90.000,E1 294.847} C_DIS
LIN {X 0.091,Y -532.745,Z 1144.429,A 0.000,B 0.000,C 90.000,E1 293.131} C_DIS
LIN {X 0.090,Y -532.751,Z 1144.419,A 0.000,B 0.000,C 90.000,E1 291.408} C_DIS
LIN {X -0.108,Y -532.619,Z 1144.411,A 0.000,B 0.000,C 90.000,E1 289.993} C_DIS
LIN {X -0.183,Y -532.329,Z 1144.405,A 0.000,B 0.000,C 90.000,E1 288.852} C_DIS
